/////////////////////////////////////digital output////////////////////////////////////////
G_IO.arDO[5].Ch[0]	:= valve_lift.extend;
G_IO.arDO[5].Ch[1]	:= valve_lift.retract;
G_IO.arDO[5].Ch[2]	:= roller_inbound.roller.forward;
G_IO.arDO[5].Ch[3]	:= roller_inbound.roller.backward;
G_IO.arDO[5].Ch[4]	:= roller_outbound.roller.forward;
G_IO.arDO[5].Ch[5]	:= roller_outbound.roller.backward;
G_IO.arDO[5].Ch[6]	:= roller_outbound_end.roller.forward;
G_IO.arDO[5].Ch[7]	:= roller_outbound_end.roller.backward;
G_IO.arDO[5].Ch[8]	:= lightcurtain_mute_left;
G_IO.arDO[5].Ch[9]	:= lightcurtain_mute_right;

G_IO.arDO[7].Ch[0]	:= valve_vacuun[0].extend;
G_IO.arDO[7].Ch[1]	:= valve_vacuun[1].extend;
G_IO.arDO[7].Ch[2]	:= valve_vacuun[2].extend;
G_IO.arDO[7].Ch[3]	:= valve_vacuun[3].extend;
G_IO.arDO[7].Ch[4]	:= valve_open_side.extend;
G_IO.arDO[7].Ch[8]	:= valve_open_side.retract;
G_IO.arDO[7].Ch[6]	:= valve_open_lift.extend;




/////////////////////////////////////axis config////////////////////////////////////////
mcAxis_lift
(
	ZSN		:=  TRUE OR st_mcAxis_lift.xHoming, //TODO link to digital input
	ZSP		:=  TRUE OR st_mcAxis_lift.xHoming, //TODO link to digital input
	IN_OUT	:= st_mcAxis_lift	, 
	AXIS	:= AxisRef_lift	, 
);
st_mcAxis_lift.bPosSensorShow	:= TRUE;
st_mcAxis_lift.bNegSensorShow	:= TRUE;
st_mcAxis_lift.rMaxAcceleration	:= 50000;
st_mcAxis_lift.rMaxDeceleration	:= 50000;
st_mcAxis_lift.rMaxJerk			:= 500000;
st_mcAxis_lift.rAcceleration	:= 2500;
st_mcAxis_lift.rDeceleration	:= 2500;
st_mcAxis_lift.rJerk			:= 12500;
st_mcAxis_lift.rMaxVelocity		:= 100;
st_mcAxis_lift.rMaxDistance		:= 50;
st_mcAxis_lift.bPosSen	:= TRUE ;//TODO link to digital input
st_mcAxis_lift.bNegSen	:= TRUE ;//TODO link to digital input
st_mcAxis_lift.mcHome.bCalibrationCam	:= TRUE;//TODO link to digital input origin
st_mcAxis_lift.bPositionSensor	:= TRUE;//TODO link to digital input origin
st_mcAxis_lift.bdirFW	:= TRUE;
st_mcAxis_lift.sNetID := '192.168.11.159.5.1';
st_mcAxis_lift.nSlaveAddr	:= 1026;

mcAxis_bag
(
	ZSN		:=  TRUE OR st_mcAxis_bag.xHoming, //TODO link to digital input
	ZSP		:=  TRUE OR st_mcAxis_bag.xHoming, //TODO link to digital input
	IN_OUT	:= st_mcAxis_bag	, 
	AXIS	:= AxisRef_bag	, 
);
st_mcAxis_bag.bPosSensorShow	:= TRUE;
st_mcAxis_bag.bNegSensorShow	:= TRUE;
st_mcAxis_bag.rMaxAcceleration	:= 50000;
st_mcAxis_bag.rMaxDeceleration	:= 50000;
st_mcAxis_bag.rMaxJerk			:= 500000;
st_mcAxis_bag.rAcceleration	:= 2500;
st_mcAxis_bag.rDeceleration	:= 2500;
st_mcAxis_bag.rJerk			:= 12500;
st_mcAxis_bag.rMaxVelocity		:= 100;
st_mcAxis_bag.rMaxDistance		:= 50;
st_mcAxis_bag.bPosSen	:= TRUE ;//TODO link to digital input
st_mcAxis_bag.bNegSen	:= TRUE ;//TODO link to digital input
st_mcAxis_bag.mcHome.bCalibrationCam	:= TRUE;//TODO link to digital input origin
st_mcAxis_bag.bPositionSensor	:= TRUE;//TODO link to digital input origin
st_mcAxis_bag.bdirFW	:= TRUE;
st_mcAxis_bag.sNetID := '192.168.11.159.5.1';
st_mcAxis_bag.nSlaveAddr	:= 1027;

mcAxis_vacuun[0]
(
	ZSN		:=  TRUE OR st_mcAxis_vacuun[0].xHoming, //TODO link to digital input
	ZSP		:=  TRUE OR st_mcAxis_vacuun[0].xHoming, //TODO link to digital input
	IN_OUT	:= st_mcAxis_vacuun[0], 
	AXIS	:= AxisRef_vacuun[0]	, 
);
st_mcAxis_vacuun[0].bPosSensorShow	:= TRUE;
st_mcAxis_vacuun[0].bNegSensorShow	:= TRUE;
st_mcAxis_vacuun[0].rMaxAcceleration	:= 50000;
st_mcAxis_vacuun[0].rMaxDeceleration	:= 50000;
st_mcAxis_vacuun[0].rMaxJerk			:= 500000;
st_mcAxis_vacuun[0].rAcceleration	:= 2500;
st_mcAxis_vacuun[0].rDeceleration	:= 2500;
st_mcAxis_vacuun[0].rJerk			:= 12500;
st_mcAxis_vacuun[0].rMaxVelocity		:= 100;
st_mcAxis_vacuun[0].rMaxDistance		:= 50;
st_mcAxis_vacuun[0].bPosSen	:= TRUE ;//TODO link to digital input
st_mcAxis_vacuun[0].bNegSen	:= TRUE ;//TODO link to digital input
st_mcAxis_vacuun[0].mcHome.bCalibrationCam	:= TRUE;//TODO link to digital input origin
st_mcAxis_vacuun[0].bPositionSensor	:= TRUE;//TODO link to digital input origin
st_mcAxis_vacuun[0].bdirFW	:= TRUE;
st_mcAxis_vacuun[0].sNetID := '192.168.11.159.5.1';
st_mcAxis_vacuun[0].nSlaveAddr	:= 1032;
st_mcAxis_vacuun[0].iAxis	:= 0;

mcAxis_vacuun[1]
(
	ZSN		:=  TRUE OR st_mcAxis_vacuun[1].xHoming, //TODO link to digital input
	ZSP		:=  TRUE OR st_mcAxis_vacuun[1].xHoming, //TODO link to digital input
	IN_OUT	:= st_mcAxis_vacuun[1]	, 
	AXIS	:= AxisRef_vacuun[1]	, 
);
st_mcAxis_vacuun[1].bPosSensorShow	:= TRUE;
st_mcAxis_vacuun[1].bNegSensorShow	:= TRUE;
st_mcAxis_vacuun[1].rMaxAcceleration	:= 50000;
st_mcAxis_vacuun[1].rMaxDeceleration	:= 50000;
st_mcAxis_vacuun[1].rMaxJerk			:= 500000;
st_mcAxis_vacuun[1].rAcceleration	:= 2500;
st_mcAxis_vacuun[1].rDeceleration	:= 2500;
st_mcAxis_vacuun[1].rJerk			:= 12500;
st_mcAxis_vacuun[1].rMaxVelocity		:= 100;
st_mcAxis_vacuun[1].rMaxDistance		:= 50;
st_mcAxis_vacuun[1].bPosSen	:= TRUE ;//TODO link to digital input
st_mcAxis_vacuun[1].bNegSen	:= TRUE ;//TODO link to digital input
st_mcAxis_vacuun[1].mcHome.bCalibrationCam	:= TRUE;//TODO link to digital input origin
st_mcAxis_vacuun[1].bPositionSensor	:= TRUE;//TODO link to digital input origin
st_mcAxis_vacuun[1].bdirFW	:= TRUE;
st_mcAxis_vacuun[1].sNetID := '192.168.11.159.5.1';
st_mcAxis_vacuun[1].nSlaveAddr	:= 1032;
st_mcAxis_vacuun[1].iAxis	:= 1;

mcAxis_bagOpen[0]
(
	ZSN		:=  TRUE OR st_mcAxis_bagOpen[0].xHoming, //TODO link to digital input
	ZSP		:=  TRUE OR st_mcAxis_bagOpen[0].xHoming, //TODO link to digital input
	IN_OUT	:= st_mcAxis_bagOpen[0]	, 
	AXIS	:= AxisRef_bagOpen[0]	, 
);
st_mcAxis_bagOpen[0].bPosSensorShow	:= TRUE;
st_mcAxis_bagOpen[0].bNegSensorShow	:= TRUE;
st_mcAxis_bagOpen[0].rMaxAcceleration	:= 50000;
st_mcAxis_bagOpen[0].rMaxDeceleration	:= 50000;
st_mcAxis_bagOpen[0].rMaxJerk			:= 500000;
st_mcAxis_bagOpen[0].rAcceleration	:= 2500;
st_mcAxis_bagOpen[0].rDeceleration	:= 2500;
st_mcAxis_bagOpen[0].rJerk			:= 12500;
st_mcAxis_bagOpen[0].rMaxVelocity		:= 100;
st_mcAxis_bagOpen[0].rMaxDistance		:= 50;
st_mcAxis_bagOpen[0].bPosSen	:= TRUE ;//TODO link to digital input
st_mcAxis_bagOpen[0].bNegSen	:= TRUE ;//TODO link to digital input
st_mcAxis_bagOpen[0].mcHome.bCalibrationCam	:= TRUE;//TODO link to digital input origin
st_mcAxis_bagOpen[0].bPositionSensor	:= TRUE;//TODO link to digital input origin
st_mcAxis_bagOpen[0].bdirFW	:= TRUE;
st_mcAxis_bagOpen[0].sNetID := '192.168.11.159.5.1';
st_mcAxis_bagOpen[0].nSlaveAddr	:= 1033;
st_mcAxis_bagOpen[0].iAxis	:= 0;

mcAxis_bagOpen[1]
(
	ZSN		:=  TRUE OR st_mcAxis_bagOpen[1].xHoming, //TODO link to digital input
	ZSP		:=  TRUE OR st_mcAxis_bagOpen[1].xHoming, //TODO link to digital input
	IN_OUT	:= st_mcAxis_bagOpen[1]	, 
	AXIS	:= AxisRef_bagOpen[1]	, 
);
st_mcAxis_bagOpen[1].bPosSensorShow	:= TRUE;
st_mcAxis_bagOpen[1].bNegSensorShow	:= TRUE;
st_mcAxis_bagOpen[1].rMaxAcceleration	:= 50000;
st_mcAxis_bagOpen[1].rMaxDeceleration	:= 50000;
st_mcAxis_bagOpen[1].rMaxJerk			:= 500000;
st_mcAxis_bagOpen[1].rAcceleration	:= 2500;
st_mcAxis_bagOpen[1].rDeceleration	:= 2500;
st_mcAxis_bagOpen[1].rJerk			:= 12500;
st_mcAxis_bagOpen[1].rMaxVelocity		:= 100;
st_mcAxis_bagOpen[1].rMaxDistance		:= 50;
st_mcAxis_bagOpen[1].bPosSen	:= TRUE ;//TODO link to digital input
st_mcAxis_bagOpen[1].bNegSen	:= TRUE ;//TODO link to digital input
st_mcAxis_bagOpen[1].mcHome.bCalibrationCam	:= TRUE;//TODO link to digital input origin
st_mcAxis_bagOpen[1].bPositionSensor	:= TRUE;//TODO link to digital input origin
st_mcAxis_bagOpen[1].bdirFW	:= TRUE;
st_mcAxis_bagOpen[1].sNetID := '192.168.11.159.5.1';
st_mcAxis_bagOpen[1].nSlaveAddr	:= 1033;
st_mcAxis_bagOpen[1].iAxis	:= 1;

mcAxis_bagOpen[2]
(
	ZSN		:=  TRUE OR st_mcAxis_bagOpen[2].xHoming, //TODO link to digital input
	ZSP		:=  TRUE OR st_mcAxis_bagOpen[2].xHoming, //TODO link to digital input
	IN_OUT	:= st_mcAxis_bagOpen[2]	, 
	AXIS	:= AxisRef_bagOpen[2]	, 
);
st_mcAxis_bagOpen[2].bPosSensorShow	:= TRUE;
st_mcAxis_bagOpen[2].bNegSensorShow	:= TRUE;
st_mcAxis_bagOpen[2].rMaxAcceleration	:= 50000;
st_mcAxis_bagOpen[2].rMaxDeceleration	:= 50000;
st_mcAxis_bagOpen[2].rMaxJerk			:= 500000;
st_mcAxis_bagOpen[2].rAcceleration	:= 2500;
st_mcAxis_bagOpen[2].rDeceleration	:= 2500;
st_mcAxis_bagOpen[2].rJerk			:= 12500;
st_mcAxis_bagOpen[2].rMaxVelocity		:= 100;
st_mcAxis_bagOpen[2].rMaxDistance		:= 50;
st_mcAxis_bagOpen[2].bPosSen	:= TRUE ;//TODO link to digital input
st_mcAxis_bagOpen[2].bNegSen	:= TRUE ;//TODO link to digital input
st_mcAxis_bagOpen[2].mcHome.bCalibrationCam	:= TRUE;//TODO link to digital input origin
st_mcAxis_bagOpen[2].bPositionSensor	:= TRUE;//TODO link to digital input origin
st_mcAxis_bagOpen[2].bdirFW	:= TRUE;
st_mcAxis_bagOpen[2].sNetID := '192.168.11.159.5.1';
st_mcAxis_bagOpen[2].nSlaveAddr	:= 1034;
st_mcAxis_bagOpen[2].iAxis	:= 0;

mcAxis_bagOpen[3]
(
	ZSN		:=  TRUE OR st_mcAxis_bagOpen[3].xHoming, //TODO link to digital input
	ZSP		:=  TRUE OR st_mcAxis_bagOpen[3].xHoming, //TODO link to digital input
	IN_OUT	:= st_mcAxis_bagOpen[3]	, 
	AXIS	:= AxisRef_bagOpen[3]	, 
);
st_mcAxis_bagOpen[3].bPosSensorShow	:= TRUE;
st_mcAxis_bagOpen[3].bNegSensorShow	:= TRUE;
st_mcAxis_bagOpen[3].rMaxAcceleration	:= 50000;
st_mcAxis_bagOpen[3].rMaxDeceleration	:= 50000;
st_mcAxis_bagOpen[3].rMaxJerk			:= 500000;
st_mcAxis_bagOpen[3].rAcceleration	:= 2500;
st_mcAxis_bagOpen[3].rDeceleration	:= 2500;
st_mcAxis_bagOpen[3].rJerk			:= 12500;
st_mcAxis_bagOpen[3].rMaxVelocity		:= 100;
st_mcAxis_bagOpen[3].rMaxDistance		:= 50;
st_mcAxis_bagOpen[3].bPosSen	:= TRUE ;//TODO link to digital input
st_mcAxis_bagOpen[3].bNegSen	:= TRUE ;//TODO link to digital input
st_mcAxis_bagOpen[3].mcHome.bCalibrationCam	:= TRUE;//TODO link to digital input origin
st_mcAxis_bagOpen[3].bPositionSensor	:= TRUE;//TODO link to digital input origin
st_mcAxis_bagOpen[3].bdirFW	:= TRUE;
st_mcAxis_bagOpen[3].sNetID := '192.168.11.159.5.1';
st_mcAxis_bagOpen[3].nSlaveAddr	:= 1034;
st_mcAxis_bagOpen[3].iAxis	:= 1;



IF MAIN.firstCycle THEN
//	st_mcAxis_bag.mcPower.Enable	:= TRUE;
	st_mcAxis_lift.mcPower.Enable	:= TRUE;	
END_IF
END_METHOD

METHOD M_reset : BOOL
VAR_INPUT
END_VAR
M_reset	:= FALSE;
ton_timeout.IN	:= FALSE;
event.sMethod	:= 'reset';
error_status	:= OrderToteErrorStatus.NO_ERROR;
IF xError THEN
	st_mcAxis_lift.mcStop.Execute	:= FALSE;
	st_mcAxis_vacuun[0].mcStop.Execute	:= FALSE;
	st_mcAxis_vacuun[1].mcStop.Execute	:= FALSE;
	st_mcAxis_bagOpen[0].mcStop.Execute	:= FALSE;
	st_mcAxis_bagOpen[1].mcStop.Execute	:= FALSE;
	st_mcAxis_bagOpen[2].mcStop.Execute	:= FALSE;
	st_mcAxis_bagOpen[3].mcStop.Execute	:= FALSE;	
	st_mcAxis_lift.mcReset.Execute			:= TRUE;
	st_mcAxis_vacuun[0].mcReset.Execute		:= TRUE;
	st_mcAxis_vacuun[1].mcReset.Execute		:= TRUE;
	st_mcAxis_bagOpen[0].mcReset.Execute	:= TRUE;
	st_mcAxis_bagOpen[1].mcReset.Execute	:= TRUE;
	st_mcAxis_bagOpen[2].mcReset.Execute	:= TRUE;
	st_mcAxis_bagOpen[3].mcReset.Execute	:= TRUE;	
	
	IF eStates<>E_WorkingStates.IDLE THEN
		eStates	:= eStateTemp;//continue
	END_IF
		
	xError	:= FALSE;
ELSE
	;
END_IF

//todo:check if reset successful
M_reset	:= TRUE;
END_METHOD

METHOD M_run : BOOL
VAR_INPUT
END_VAR
//
IF M_checkCondition(condition:= E_Condition.NO_TOTE) THEN
	;
END_IF
//check no tote of working
//wait new tote of loading
//tote load
END_METHOD

METHOD M_runStart : BOOL
VAR_INPUT
END_VAR
M_runStart	:= FALSE;

st_mcAxis_vacuun[0].mcPower.Enable	:= TRUE;	
st_mcAxis_vacuun[1].mcPower.Enable	:= TRUE;
st_mcAxis_bagOpen[0].mcPower.Enable	:= TRUE;
st_mcAxis_bagOpen[1].mcPower.Enable	:= TRUE;
st_mcAxis_bagOpen[2].mcPower.Enable	:= TRUE;
st_mcAxis_bagOpen[3].mcPower.Enable	:= TRUE;

st_mcAxis_lift.mcPower.Enable	:= TRUE;

current_tote_status	:= ToteStatus.UNKNOWN;

M_checkCondition(condition:=E_Condition.TOTE_READY);

IF st_mcAxis_vacuun[0].mcReadStatus.StandStill AND st_mcAxis_vacuun[1].mcReadStatus.StandStill AND st_mcAxis_bagOpen[0].mcReadStatus.StandStill
AND st_mcAxis_bagOpen[1].mcReadStatus.StandStill AND st_mcAxis_bagOpen[2].mcReadStatus.StandStill AND st_mcAxis_bagOpen[3].mcReadStatus.StandStill 
AND st_mcAxis_lift.mcReadStatus.StandStill THEN
	M_runStart	:= TRUE;
END_IF	

M_runStart	:= TRUE;
END_METHOD

METHOD M_safetyEvent : BOOL
VAR_INPUT
END_VAR
M_safetyEvent	:= FALSE;

roller_inbound.roller.forward			:= FALSE;
roller_inbound.roller.backward			:= FALSE;
roller_outbound.roller.forward			:= FALSE;
roller_outbound.roller.backward			:= FALSE;
roller_outbound_end.roller.forward		:= FALSE;	
roller_outbound_end.roller.backward		:= FALSE;	

st_mcAxis_vacuun[0].mcMoveAbsolute.Execute	:= FALSE;
st_mcAxis_vacuun[1].mcMoveAbsolute.Execute	:= FALSE;
st_mcAxis_bagOpen[0].mcMoveAbsolute.Execute	:= FALSE;
st_mcAxis_bagOpen[1].mcMoveAbsolute.Execute	:= FALSE;
st_mcAxis_bagOpen[2].mcMoveAbsolute.Execute	:= FALSE;
st_mcAxis_bagOpen[3].mcMoveAbsolute.Execute	:= FALSE;
st_mcAxis_lift.mcMoveAbsolute.Execute	:= FALSE;	

st_mcAxis_vacuun[0].mcStop.Execute	:= TRUE;
st_mcAxis_vacuun[1].mcStop.Execute	:= TRUE;
st_mcAxis_bagOpen[0].mcStop.Execute	:= TRUE;
st_mcAxis_bagOpen[1].mcStop.Execute	:= TRUE;
st_mcAxis_bagOpen[2].mcStop.Execute	:= TRUE;
st_mcAxis_bagOpen[3].mcStop.Execute	:= TRUE;


st_mcAxis_lift.mcStop.Execute	:= TRUE;

M_safetyEvent	:= TRUE;
END_METHOD

METHOD M_toteLoad : BOOL
VAR_INPUT
END_VAR
M_toteLoad	:= FALSE;
IF roller_inbound.photo_sensor.Q THEN
	roller_inbound.roller.forward	:= FALSE;
	ADSLOGSTR(msgCtrlMask:= ADSLOG_MSGTYPE_LOG,msgFmtStr:='tote load finish',strArg:='MSG ARG');
ELSE
	roller_inbound.roller.forward	:= TRUE;
	ADSLOGSTR(msgCtrlMask:= ADSLOG_MSGTYPE_LOG,msgFmtStr:='tote load start',strArg:='MSG ARG');
	M_toteLoad	:= TRUE;
END_IF
END_METHOD

METHOD M_toteUnload : BOOL
VAR_INPUT
END_VAR
M_toteUnload	:= FALSE;

CASE eStates OF 
		E_WorkingStates.TOTE_LIFT_UP:
			valve_lift.extend	:= TRUE;
			valve_lift.retract	:= FALSE;
			IF valve_lift.extended AND NOT valve_lift.retracted THEN
				eStates	:= E_WorkingStates.TOTE_UNLOAD;
			END_IF
		E_WorkingStates.TOTE_OUT:
			IF roller_outbound.photo_sensor.Q THEN
				roller_outbound.roller.forward	:= FALSE;
				M_toteUnload	:= TRUE;
			ELSE
				roller_outbound.roller.forward	:= TRUE;
			END_IF	
		E_WorkingStates.TOTE_LIFT_DOWN:	
			valve_lift.extend	:= FALSE;
			valve_lift.retract	:= TRUE;
			IF NOT valve_lift.extended AND valve_lift.retracted THEN
				M_toteUnload	:= TRUE;
			END_IF	
END_CASE
END_METHOD

METHOD M_unload : BOOL
VAR_INPUT
END_VAR
VAR_OUTPUT 

END_VAR
//initialize
//bag_open lift up & bag_open_home
//tote lift up
//outbound
//tote lift down
//done
M_unload := FALSE;
event.sMethod	:= 'unload';
//////////////////////////////////////////////////////////timeout//////////////////////////////////////////
iStateTemp	:= eStateTemp;
sStateTemp	:= INT_TO_STRING(iStateTemp);
ton_timeout();
IF eStates<>E_WorkingStates.IDLE AND eStates<>E_WorkingStates.ERROR  THEN
	IF eStateTemp=eStates THEN
		ton_timeout.IN	:=TRUE;
	ELSE
		ton_timeout.IN	:=FALSE;
		IF GVL.bAck_stop THEN
			roller_outbound.roller.forward	:= FALSE;
			roller_outbound_end.roller.forward	:= FALSE;
			RETURN;		
		END_IF
		eStateTemp	:= eStates;
	END_IF
ELSE
	ton_timeout.IN	:=FALSE;
END_IF
IF ton_timeout.Q THEN	
	ton_timeout.IN	:=FALSE;
	CASE eStates OF
	
		E_WorkingStates.WAIT_UNLOADING://wait signal from logtech and app to unload the tote
			;
		E_WorkingStates.BAG_OPEN_UP:	
			event.sEventType	:= 'error';
			event.sEvent_MSG	:= CONCAT('BAG_OPEN_UP ','timeout');
			event.sStepID		:= sStateTemp;
		E_WorkingStates.BAG_CLOSE:	
			event.sEventType	:= 'error';
			event.sEvent_MSG	:= CONCAT('BAG_CLOSE or TOTE_LIFT_UP ','timeout');
			event.sStepID		:= sStateTemp;						
		E_WorkingStates.TOTE_LIFT_UP:
			event.sEventType	:= 'error';
			event.sEvent_MSG	:= CONCAT('TOTE_LIFT_UP ','timeout');
			event.sStepID		:= sStateTemp;
		E_WorkingStates.TOTE_UNLOAD:
			event.sEventType	:= 'error';
			event.sEvent_MSG	:= CONCAT('TOTE_UNLOAD ','timeout');
			event.sStepID		:= sStateTemp;

		E_WorkingStates.WAIT_SENSOR_OFF:	
			event.sEventType	:= 'error';
			event.sEvent_MSG	:= CONCAT('WAIT_SENSOR_OFF ','timeout');
			event.sStepID		:= sStateTemp;	
		E_WorkingStates.TOTE_LIFT_DOWN:
			event.sEventType	:= 'error';
			event.sEvent_MSG	:= CONCAT('TOTE_LIFT_DOWN ','timeout');
			event.sStepID		:= sStateTemp;
		ELSE
			event.sEventType	:= 'error';
			event.sEvent_MSG	:= CONCAT('unknow estate ','timeout');
			event.sStepID		:= sStateTemp;			
	END_CASE
	IF eStates<>E_WorkingStates.IDLE AND eStates<>E_WorkingStates.WAIT_UNLOADING AND eStates<>E_WorkingStates.BAG_OPEN_UP THEN
		eStates	:= E_WorkingStates.ERROR;
		error_status	:= OrderToteErrorStatus.MECHANICAL_ERROR;
		Event_add(event);
	END_IF
	
END_IF

CASE eStates OF 
		E_WorkingStates.IDLE:
			
			ton_timeout.PT	:= T#3S;
			xLoading	:= FALSE;
			xUnloading	:= FALSE;
			eStates	:= E_WorkingStates.INIT;
		E_WorkingStates.INIT:	
			ADSLOGSTR(msgCtrlMask:= ADSLOG_MSGTYPE_LOG,msgFmtStr:='unload start',strArg:='');
			xUnloading	:= TRUE;
			st_mcAxis_vacuun[0].mcMoveAbsolute.Execute	:= FALSE;
			st_mcAxis_vacuun[1].mcMoveAbsolute.Execute	:= FALSE;
			st_mcAxis_bagOpen[0].mcMoveAbsolute.Execute	:= FALSE;
			st_mcAxis_bagOpen[1].mcMoveAbsolute.Execute	:= FALSE;
			st_mcAxis_bagOpen[2].mcMoveAbsolute.Execute	:= FALSE;
			st_mcAxis_bagOpen[3].mcMoveAbsolute.Execute	:= FALSE;			
	
			st_mcAxis_lift.mcMoveAbsolute.Execute	:= FALSE;
			eStates	:= E_WorkingStates.WAIT_UNLOADING;
		E_WorkingStates.WAIT_UNLOADING://wait signal from logtech and app to unload the tote
			workflow_status	:= ToteSubsystemWorkflowStatus.WAITING_FOR_UNLOADING;
			tote_status	:= ToteStatus.READY;
			eStates	:= E_WorkingStates.BAG_OPEN_UP;	
			
//		E_WorkingStates.BAG_OPEN_AXIS_CYCLINDER_UP:
//			ton_timeout.PT	:= T#1S;
//			valve_open_lift.extend	:= FALSE;
//			valve_open_lift.retract	:= TRUE;
//			IF NOT valve_open_lift.extended AND valve_open_lift.retracted THEN
//				eStates	:= E_WorkingStates.BAG_OPEN_UP;
//			END_IF
//			IF ton_timeout.Q THEN
//				eStates	:= E_WorkingStates.BAG_OPEN_UP;
//			END_IF
		E_WorkingStates.BAG_OPEN_UP:	
			ton_timeout.PT	:= T#1S;
			valve_open_lift.extend	:= FALSE;
			valve_open_lift.retract	:= TRUE;			
			workflow_status	:= ToteSubsystemWorkflowStatus.OUTBOUNDING;	
			tote_status	:= ToteStatus.LOADED;		
			st_mcAxis_lift.mcMoveAbsolute.Execute	:= TRUE;		
			st_mcAxis_lift.rActualPosSet	:= rPos_lift_up;
			st_mcAxis_lift.rVelocitySet	:= 250;
			IF st_mcAxis_lift.mcMoveAbsolute.Done 
			AND ((NOT valve_open_lift.extended AND valve_open_lift.retracted) OR ton_timeout.Q) THEN
				eStates	:= E_WorkingStates.BAG_OPEN_HOME;
			END_IF	
		E_WorkingStates.BAG_OPEN_HOME:	
			ton_timeout.PT	:= T#5S;
			valve_open_side.extend	:= FALSE;
			valve_open_side.retract	:= TRUE;		
			st_mcAxis_vacuun[0].mcMoveAbsolute.Execute	:= TRUE;		
			st_mcAxis_vacuun[0].rActualPosSet	:= rPos_vacuun_working[0];
			st_mcAxis_vacuun[0].rVelocitySet	:= 450;
			st_mcAxis_vacuun[1].mcMoveAbsolute.Execute	:= TRUE;		
			st_mcAxis_vacuun[1].rActualPosSet	:= rPos_vacuun_working[1];
			st_mcAxis_vacuun[1].rVelocitySet	:= 450;			
			st_mcAxis_bagOpen[0].mcMoveAbsolute.Execute	:= TRUE;		
			st_mcAxis_bagOpen[0].rActualPosSet	:= rPos_bag_begin[0];
			st_mcAxis_bagOpen[0].rVelocitySet	:= 200;			
			st_mcAxis_bagOpen[1].mcMoveAbsolute.Execute	:= TRUE;		
			st_mcAxis_bagOpen[1].rActualPosSet	:= rPos_bag_begin[1];
			st_mcAxis_bagOpen[1].rVelocitySet	:= 200;				
			st_mcAxis_bagOpen[2].mcMoveAbsolute.Execute	:= TRUE;		
			st_mcAxis_bagOpen[2].rActualPosSet	:= rPos_bag_begin[2];
			st_mcAxis_bagOpen[2].rVelocitySet	:= 200;				
			st_mcAxis_bagOpen[3].mcMoveAbsolute.Execute	:= TRUE;		
			st_mcAxis_bagOpen[3].rActualPosSet	:= rPos_bag_begin[3];
			st_mcAxis_bagOpen[3].rVelocitySet	:= 200;		
			valve_lift.extend	:= TRUE;
			valve_lift.retract	:= FALSE;				
			IF st_mcAxis_vacuun[0].mcMoveAbsolute.Done AND st_mcAxis_vacuun[1].mcMoveAbsolute.Done 
			AND st_mcAxis_bagOpen[0].mcMoveAbsolute.Done AND st_mcAxis_bagOpen[1].mcMoveAbsolute.Done 
			AND st_mcAxis_bagOpen[2].mcMoveAbsolute.Done AND st_mcAxis_bagOpen[3].mcMoveAbsolute.Done 
			AND(NOT valve_open_side.extended AND valve_open_side.retracted) 
			AND (valve_lift.extended AND NOT valve_lift.retracted) THEN
				st_mcAxis_vacuun[0].mcMoveAbsolute.Execute	:= FALSE;
				st_mcAxis_vacuun[1].mcMoveAbsolute.Execute	:= FALSE;
				st_mcAxis_bagOpen[0].mcMoveAbsolute.Execute	:= FALSE;
				st_mcAxis_bagOpen[1].mcMoveAbsolute.Execute	:= FALSE;
				st_mcAxis_bagOpen[2].mcMoveAbsolute.Execute	:= FALSE;
				st_mcAxis_bagOpen[3].mcMoveAbsolute.Execute	:= FALSE;
				eStates	:= E_WorkingStates.TOTE_UNLOAD;
			END_IF								
	
//		E_WorkingStates.BAG_CLOSE:	
//			st_mcAxis_bag.mcMoveAbsolute.Execute	:= TRUE;		
//			st_mcAxis_bag.rActualPosSet	:= rPos_bag_closed;
//			st_mcAxis_bag.rVelocitySet	:= 250;
//			valve_lift.extend	:= TRUE;
//			valve_lift.retract	:= FALSE;
//			IF st_mcAxis_bag.mcMoveAbsolute.Done AND valve_lift.extended AND NOT valve_lift.retracted THEN
//				st_mcAxis_bag.mcMoveAbsolute.Execute	:= FALSE;
//				eStates	:= E_WorkingStates.TOTE_UNLOAD;
//			END_IF							
//		E_WorkingStates.TOTE_LIFT_UP:
//			ton_timeout.PT	:= T#3S;
//			valve_lift.extend	:= TRUE;
//			valve_lift.retract	:= FALSE;
//			IF valve_lift.extended AND NOT valve_lift.retracted THEN
//				eStates	:= E_WorkingStates.TOTE_UNLOAD;
//			END_IF
		E_WorkingStates.TOTE_UNLOAD:
			ton_timeout.PT	:= T#5S;
			roller_outbound.roller.forward		:= TRUE;
			roller_outbound_end.roller.forward	:= TRUE;
			IF roller_outbound.photo_sensor.Q THEN
				eStates	:= E_WorkingStates.WAIT_SENSOR_OFF;			
			END_IF	
		E_WorkingStates.WAIT_SENSOR_OFF:
			roller_outbound.roller.forward		:= TRUE;
			roller_outbound_end.roller.forward	:= TRUE;	
			IF NOT roller_outbound.photo_sensor.Q THEN
				roller_outbound.roller.forward		:= FALSE;	
				roller_outbound_end.roller.forward	:= FALSE;
				eStates	:= E_WorkingStates.TOTE_LIFT_DOWN;			
			END_IF			
		E_WorkingStates.TOTE_LIFT_DOWN:
			ton_timeout.PT	:= T#3S;	
			valve_lift.extend	:= FALSE;
			valve_lift.retract	:= TRUE;
			IF NOT valve_lift.extended AND valve_lift.retracted THEN
				eStates	:= E_WorkingStates.DONE;
			END_IF				
		E_WorkingStates.DONE:	
			ADSLOGSTR(msgCtrlMask:= ADSLOG_MSGTYPE_LOG,msgFmtStr:='unload end',strArg:='');
			workflow_status	:= ToteSubsystemWorkflowStatus.IDLE;
			tote_status	:= ToteStatus.EMPTY;			
			M_unload	:= TRUE;
			xUnloading	:= FALSE;
			eStates	:= E_WorkingStates.IDLE;
		E_WorkingStates.ERROR:
			xError	:=	TRUE;
			workflow_status	:= ToteSubsystemWorkflowStatus.IDLE;
			roller_outbound.roller.forward		:= FALSE;	
			roller_outbound_end.roller.forward	:= FALSE;
			st_mcAxis_vacuun[0].mcMoveAbsolute.Execute	:= FALSE;
			st_mcAxis_vacuun[1].mcMoveAbsolute.Execute	:= FALSE;
			st_mcAxis_bagOpen[0].mcMoveAbsolute.Execute	:= FALSE;
			st_mcAxis_bagOpen[1].mcMoveAbsolute.Execute	:= FALSE;
			st_mcAxis_bagOpen[2].mcMoveAbsolute.Execute	:= FALSE;
			st_mcAxis_bagOpen[3].mcMoveAbsolute.Execute	:= FALSE;			
			st_mcAxis_lift.mcMoveAbsolute.Execute	:= FALSE;
			M_unload 		:= TRUE;

		
END_CASE
END_METHOD

METHOD M_waitCondition : BOOL
VAR_INPUT
	condition	: E_Condition;
END_VAR
M_waitCondition	:= FALSE;
CASE condition OF
	E_Condition.NO_TOTE:
	 	IF NOT roller_inbound.photo_sensor.Q THEN
			M_waitCondition	:= TRUE;
		END_IF
	E_Condition.TOTE_IN:
	 	IF roller_inbound.photo_sensor.Q THEN
			M_waitCondition	:= TRUE;
		END_IF	
	E_Condition.READY_LOADING_TOTE:
		IF (pre_tote_status=ToteStatus.READY AND GVL.fb_loading.eTransfer=E_Transfer.UNLOAD) OR tote_status=ToteStatus.LOADED THEN
			M_waitCondition	:= TRUE;
		END_IF	
END_CASE
END_METHOD

END_FUNCTION_BLOCK

// ---- Mian/machine/axis/FB_MotionAxis_MC.TcPOU
FUNCTION_BLOCK FB_MotionAxis_MC

VAR_INPUT
	ZSN	   			: BOOL												;
	ZSP				: BOOL												; 
	Exceeding_us			: INT;
	sNameAxis				: STRING [40];

END_VAR         	
                	
VAR  
	rtFirstCycle	: R_TRIG;						
	mcHomeAxis		: 	MC_HomeAxis						;//ADD BY EVAN 
	sAxisName		: STRING											;//Axis name          	
	xPlus			: BOOL												;	
	xMinus			: BOOL												;
	bDone			: BOOL												;	

// Variables for Hard Stop Homing	                        			
	iStatehsHomig	: E_HomingSteps := E_HomingSteps.IDLE				;
	rtHome			: R_TRIG											;
	rtHomeReset		: R_TRIG											;
	tonTimeOut		: TON												;
	xTimerStart		: BOOL												;
	bLSDefaultVal	: BOOL												; // Save Def value from driver
	xHomeError		: BOOL												;
// Variables for Force Control          					

	rtForceC		: R_TRIG											;
	rtForceCReset	: R_TRIG											;
	DelMaxPos		: LREAL 											;
	rCurrLimit		: LREAL												;
	StartPos		: LREAL												;
	xForceCError	: BOOL												;
//	Variables for Backlash Compensation
	rLastMove		: LREAL := 1										;
	tonBackComp		: TON												;
	rBacklashPer	: LREAL												;	
	
// Variables for errors
	rtError					:	R_TRIG;
	pTextType				:	POINTER TO STRING;
	sAxisErrorID			:	STRING(10);	
	ErrorMSG				:	STRING[255];

//	Exceeding time measuring
	sysTime					:	GETCPUCOUNTER;//GETSYSTEMTIME;					//	Used to measure execution time.
	uStartTime				:	UDINT;
	uFinishTime				:	UDINT;
	ftimeDiff				:	REAL;
	ton_dly	: TON;
	offset	: WORD;
END_VAR         	
                	
VAR_IN_OUT      	
	IN_OUT 			: ST_MotionAxis_MC	;//struct for each axis
	AXIS 			: AXIS_REF			;//Axis obj	
END_VAR

VAR_OUTPUT
	xError			: BOOL				;
	xBusy			: BOOL				;
END_VAR
VAR CONSTANT
	parallelGroupTLName		:	STRING := 'Port_851.TL_Axis_Error';
END_VAR

(* Power options ********************************************************************************************)			
IN_OUT.mcPower(
	Axis				:= AXIS, 
	Enable				:= , 
	Enable_Positive		:= ZSP, 
	Enable_Negative		:= ZSN OR IN_OUT.mcHome.Busy, 
	Override			:= , 
	BufferMode			:= , 
	Options				:= , 
	Status				=> , 
	Busy				=> , 
	Active				=> , 
	Error				=> , 
	ErrorID				=> );
	
(* Halt Mode ********************************************************************************************)	
IN_OUT.mcHalt(
	Axis				:= AXIS, 
	Execute				:= , 
	Deceleration		:= IN_OUT.rDeceleration, 
	Jerk				:= , 
	BufferMode			:= , 
	Options				:= , 
	Done				=> , 
	Busy				=> , 
	Active				=> , 
	CommandAborted		=> , 
	Error				=> , 
	ErrorID				=> );
	
(* Homing ***********************************************************************************************)
IN_OUT.mcHome(
	Axis				:= AXIS, 
	Execute				:= , 
	Position			:= in_out.rFirstpos, 
	HomingMode			:= MC_Direct, 
	BufferMode			:= , 
	Options				:= , 
	bCalibrationCam		:= ,//NOT  ZSN, 
	Done				=> , 
	Busy				=> , 
	Active				=> , 
	CommandAborted		=> , 
	Error				=> , 
	ErrorID				=> );
	
(* JOG **************************************************************************************************)
IN_OUT.mcJog(
	Axis				:= AXIS, 
	JogForward			:= , 
	JogBackwards		:= , 
	Mode				:= E_JogMode.MC_JOGMODE_CONTINOUS, 
	Position			:= , 
	Velocity			:= IN_OUT.rVelocity, 
	Acceleration		:= IN_OUT.rAcceleration, 
	Deceleration		:= IN_OUT.rDeceleration, 
	Jerk				:= IN_OUT.rJerk, 
	Done				=> , 
	Busy				=> , 
	Active				=> , 
	CommandAborted		=> , 
	Error				=> , 
	ErrorID				=> );
	
(* Move Absolute ****************************************************************************************)	
IN_OUT.mcMoveAbsolute(
	Axis				:= AXIS, 
	Execute				:= , 
	Position			:= IN_OUT.rActualPosSet, 
	Velocity			:= IN_OUT.rVelocitySet,     
	Acceleration		:= IN_OUT.rAcceleration, 
	Deceleration		:= IN_OUT.rDeceleration, 
	Jerk				:= IN_OUT.rJerk,         
	BufferMode			:= , 
	Options				:= , 
	Done				=> , 
	Busy				=> , 
	Active				=> , 
	CommandAborted		=> , 
	Error				=> , 
	ErrorID				=> );

	IF IN_OUT.bMoveAbsHMI THEN
		IN_OUT.mcMoveAbsolute.Execute	:= TRUE;
		IN_OUT.rActualPosSet	:= IN_OUT.rActualPosHMI;
		IN_OUT.rVelocitySet		:= IN_OUT.rVeloPers;
	END_IF
(* Move Relative *********************************************************************************************************)
IN_OUT.mcMoveRelative(
	Axis				:= AXIS, 
	Execute				:= , 
	Distance			:= IN_OUT.rPosition + IN_OUT.rBacklashvalue, 
	Velocity			:= IN_OUT.rVelocity,      
	Acceleration		:= IN_OUT.rAcceleration,  
	Deceleration		:= IN_OUT.rDeceleration,  
	Jerk				:= IN_OUT.rJerk,          
	BufferMode			:= ,
	Options				:= , 
	Done				=> bDone, 
	Busy				=> , 
	Active				=> , 
	CommandAborted		=> , 
	Error				=> , 
	ErrorID				=> );
	
(* Move Velocity *********************************************************************************************************)
	
IN_OUT.mcMoveVelocity(
	Axis				:=	AXIS,
	Execute				:=	,
	Velocity			:=	IN_OUT.rVelocity,
	Acceleration		:=	IN_OUT.rAcceleration,
	Deceleration		:=	IN_OUT.rDeceleration,
	Jerk				:=	IN_OUT.rJerk,
	Direction			:=	IN_OUT.axisDirection,
	BufferMode			:=	,
	Options				:=	,
	InVelocity			=>	,
	Busy				=>	,
	Active				=>	,
	CommandAborted		=>	,
	Error				=>	,
	ErrorID				=>	);
	
(**)	
IN_OUT.mcReadStatus(
	Axis				:= AXIS, 
	Enable				:= TRUE, 
	Valid				=> , 
	Busy				=> , 
	Error				=> , 
	ErrorID				=> , 
	ErrorStop			=> , 
	Disabled			=> , 
	Stopping			=> , 
	StandStill			=> , 
	DiscreteMotion		=> , 
	ContinuousMotion	=> , 
	SynchronizedMotion	=> , 
	Homing				=> , 
	ConstantVelocity	=> , 
	Accelerating		=> , 
	Decelerating		=> , 
	Status				=> );
	
(* Reset ************************************************************************************************)
IN_OUT.mcReset(
	Axis				:= AXIS, 
	Execute				:= , 
	Done				=> , 
	Busy				=> , 
	Error				=> , 
	ErrorID				=> );
	
(* Stop *************************************************************************************************)
IN_OUT.mcStop(
	Axis				:= AXIS, 
	Execute				:= , 
	Deceleration		:= , 
	Jerk				:= , 
	Options				:= , 
	Done				=> , 
	Busy				=> , 
	Active				=> , 
	CommandAborted		=> , 
	Error				=> , 
	ErrorID				=> );

(* Set Position *************************************************************************************************)
in_out.mcSetpoint(
	Axis			 := AXIS, 
	Execute			 := , 
	Position		 := IN_OUT.rSetPos, 
	Mode			 := , 
	Options			 := , 
	Done			 => , 
	Busy			 => , 
	Error			 => , 
	ErrorID			 => );


(* write status *************************************************************************************************)
IN_OUT.mcWriteBoolParameter(
	Axis			:= 	AXIS, 
	Execute:= 				, 
	ParameterNumber:= 		, 
	Value:= , 
	Done=> , 
	Busy=> , 
	Error=> , 
	ErrorID=> );

(* Read status *************************************************************************************************)
IN_OUT.mcReadBoolParameter(
	Axis:= AXIS, 
	Enable:= , 
	ParameterNumber:= , 
	ReadMode:= , 
	Valid=> , 
	Busy=> , 
	Error=> , 
	ErrorID=> , 
	Value=> );	

(*Read Actualposition***************************************************************)
IN_OUT.mcReadActualPosition(
	Axis:= AXIS, 
	Enable:= TRUE, 
	Valid=> , 
	Busy=> , 
	Error=> , 
	ErrorID=> , 
	Position=> IN_OUT.rActualPos );   
(*COE write**************************************************************************)	

IN_OUT.CoeWrt(
	sNetId:= IN_OUT.sNetID, 
	nSlaveAddr:= IN_OUT.nSlaveAddr, 
	nSubIndex:= IN_OUT.nSubIndex, 
	nIndex:= IN_OUT.nIndex, 
	pSrcBuf:= ADR(IN_OUT.iSdoWrite), 
	cbBufLen:= SIZEOF(IN_OUT.iSdoWrite), 
	bExecute:= , 
	tTimeout:= , 
	bBusy=> , 
	bError=> , 
	nErrId=> );
	ton_dly(PT:=T#100MS);


offset	:= 16#800*IN_OUT.iAxis;	
CASE IN_OUT.iCoeWrt OF 
	0:
		IN_OUT.CoeWrt.bExecute := FALSE;
	1:
		IN_OUT.CoeWrt.bExecute := TRUE;
		IN_OUT.nIndex	:= 16#2005+offset;
		IN_OUT.nSubIndex	:= 16#1F;
		IN_OUT.iSdoWrite	:= 6;//clear encoder and set current position as origin
		IN_OUT.iCoeWrt	:= 10;
	2:
		IN_OUT.CoeWrt.bExecute := TRUE;
		IN_OUT.nIndex	:= 16#2002+offset;
		IN_OUT.nSubIndex	:= 16#02;
		IN_OUT.iSdoWrite	:= 1;//linear mode
		IN_OUT.iCoeWrt	:= 10;
	3:
		IN_OUT.CoeWrt.bExecute := TRUE;
		IN_OUT.nIndex	:= 16#2002+offset;
		IN_OUT.nSubIndex	:= 16#02;
		IN_OUT.iSdoWrite	:= 2;//rotate mode
		IN_OUT.iCoeWrt	:= 10;
	4:
		IN_OUT.CoeWrt.bExecute := TRUE;
		IN_OUT.nIndex	:= 16#2004+offset;
		IN_OUT.nSubIndex	:= 16#06;
		IN_OUT.iSdoWrite	:= 1;//breaker on
		IN_OUT.iCoeWrt	:= 10;
	5:
		IN_OUT.CoeWrt.bExecute := TRUE;
		IN_OUT.nIndex	:= 16#2004+offset;
		IN_OUT.nSubIndex	:= 16#06;
		IN_OUT.iSdoWrite	:= 0;//breaker off
		IN_OUT.iCoeWrt	:= 10;		
	10:		
		IN_OUT.iCoeWrt	:= 0;
END_CASE







	(*mcHomeAxis***************************************************************)
	mcHomeAxis(
		xExecute:= , 
		xReset:= , 
		InOut:=IN_OUT , 
		xRedy=> , 
		xBusy=> , 
		xDone=> , 
		xError=> ); 
	                                                                                                              	
(******************************************************************************************************************)
	
(**error flag**)

	IN_OUT.xTorqueErr	:=ABS(IN_OUT.rActTorque)>IN_OUT.rToqueLimitSet ;

	
	

	xError := IN_OUT.mcReadStatus.Error OR xHomeError OR IN_OUT.mcMoveAbsolute.Error OR IN_OUT.xTorqueErr ;	
	rtError(CLK:= (IN_OUT.mcReadStatus.ErrorID <> 0 OR xError) AND NOT IN_OUT.xMuteAxisErrorMessages);
	
(*************************** READ ERROR FROM DRIVE *************************)
rtFirstCycle(CLK:= TRUE);
sysTime(cpuCntLoDW => uStartTime);	
sysTime(cpuCntLoDW => uFinishTime);
//M_CheckExceedingTime();

(*************************** GET AXIS ERROR MESSAGE *************************)	
	
	IF rtError.Q THEN
		IF IN_OUT.xTorqueErr THEN
			sAxisErrorID	:= 'TORQUE';
		ELSE
			sAxisErrorID	:=	TO_STRING(IN_OUT.mcReadStatus.ErrorID);
		END_IF
		IN_OUT.mcStop.Execute	:= TRUE;
	
	END_IF
(**remember the Velocity**) 
	IF IN_OUT.rVeloPers <> 0 THEN 
		IN_OUT.rVelocity:= IN_OUT.rVeloPers;
	ELSE 
		IN_OUT.rVeloPers := IN_OUT.rVelocity;	
	END_IF	
(**remember the Acceleration**)
	IF IN_OUT.rAccPers <> 0 THEN 
		IN_OUT.rAcceleration:= IN_OUT.rAccPers;
	ELSE 
		IN_OUT.rAccPers := IN_OUT.rAcceleration;		
	END_IF	
(**remember the Deceleration**)
	IF IN_OUT.rDecPers <> 0 THEN 
		IN_OUT.rDeceleration:= IN_OUT.rDecPers;
	ELSE 
		IN_OUT.rDecPers := IN_OUT.rDeceleration;		
	END_IF
(**False all Executions if function done or error**)
	IF IN_OUT.mcMoveRelative.Done OR IN_OUT.mcMoveRelative.Error OR IN_OUT.mcReset.Busy THEN 
		IN_OUT.mcMoveRelative.Execute := FALSE;
	END_IF

	IF IN_OUT.mcMoveVelocity.Error OR IN_OUT.mcReset.Busy OR IN_OUT.mcMoveVelocity.Busy THEN 
		IN_OUT.mcMoveVelocity.Execute := FALSE;
	END_IF
	
	IF IN_OUT.mcSetpoint.done OR IN_OUT.mcSetpoint.Error THEN
		IN_OUT.mcSetpoint.Execute := FALSE;
	END_IF
	
    IF  IN_OUT.mcMoveAbsolute.Done OR IN_OUT.mcMoveAbsolute.Error OR IN_OUT.mcReset.Busy THEN 
		IN_OUT.mcMoveAbsolute.Execute := FALSE;
	END_IF
 
	 IF IN_OUT.mcHome.Done OR IN_OUT.mcHome.Error THEN 
		IN_OUT.mcHome.Execute := FALSE;
	END_IF
	
	IF IN_OUT.mcStop.Done OR IN_OUT.mcStop.Error THEN 
		IN_OUT.mcStop.Execute := FALSE;
	END_IF
	
	IF IN_OUT.mcReset.Done OR IN_OUT.mcReset.Error THEN 
		IN_OUT.mcReset.Execute := FALSE;
	END_IF
			
	IF IN_OUT.mcReadBoolParameter.Valid OR IN_OUT.mcReadBoolParameter.Error THEN 
		IN_OUT.mcReadBoolParameter.Enable := FALSE;
	END_IF	
	
	IF IN_OUT.mcWriteBoolParameter.Done OR IN_OUT.mcWriteBoolParameter.Error THEN 
		IN_OUT.mcWriteBoolParameter.Execute	:= FALSE;
	END_IF	
		

	
	
	
(**Save done state into temp variable**)	
	
	IF IN_OUT.mcMoveAbsolute.Done THEN
		IN_OUT.xMoveABSDone := TRUE;
	END_IF	
	
	IF IN_OUT.mcMoveRelative.Done THEN
		IN_OUT.xMoveRelDone := TRUE;
	END_IF

PROPERTY P_AxisName : STRING
SET
sAxisName := P_AxisName;
END_SET
END_PROPERTY

PROPERTY P_CurrLimit : LREAL
SET
rCurrLimit := P_CurrLimit;
END_SET
END_PROPERTY

PROPERTY P_DelMaxPos : LREAL
SET
DelMaxPos := P_DelMaxPos;
END_SET
END_PROPERTY

PROPERTY P_ForceCError : BOOL
GET
P_ForceCError := xForceCError;
END_GET
END_PROPERTY

PROPERTY P_hsHomingError : BOOL
GET
P_hsHomingError := xHomeError;
END_GET
END_PROPERTY

PROPERTY P_StartPos : LREAL
SET
StartPos := P_StartPos;
END_SET
END_PROPERTY

END_FUNCTION_BLOCK

// ---- Mian/machine/loading moudle/FB_loading.TcPOU
FUNCTION_BLOCK FB_loading
VAR_INPUT
	pre_tote_status			: ToteStatus;//roller -1 totestatus=ready
	next_tote_status		: ToteStatus;//roller +1 totestatus=empty
	bRun					: BOOL;
	bReset					: BOOL;
	bSafety					: BOOL;
	lightTower				: ST_LightTower;
END_VAR
VAR_OUTPUT
	ready_recive		: BOOL;
	tote_recivied_current		: BOOL;//current roller recived the tote
END_VAR
VAR
	current_tote_status	: ToteStatus;
	ton_timeout			: TON;	
	eStates				: E_LoadingStates := E_LoadingStates.IDLE;
	eStateTemp			: E_LoadingStates := E_LoadingStates.IDLE;
	iStateTemp			: INT;
	sStateTemp			: STRING;
	errorMessage		: STRING;
	xError				: BOOL;
	event				: ST_EVENT;
	rt_error			: R_TRIG;
	eTransfer			: E_Transfer;
///////////////hardware define//////////////////	
	roller_x					: Roller_x;
	roller_y					: Roller_y;
	photo_sensor_tote_detection	: FB_DigitalInput;
	EDM_KA7						: BOOL;
	floodlight					: BOOL;
	mcAxis	 					: FB_MotionAxis_MC;
	st_mcAxis					: ST_MotionAxis_MC;
	AxisRef						: AXIS_REF;	
END_VAR
VAR CONSTANT
	rPos_load	: REAL := 0;
	rPos_unload	: REAL := 1;
	sComponent_name			: STRING := 'fb_loading';
END_VAR

M_mapping();


rt_error(CLK:=(roller_x.roller.err OR roller_y.roller.err OR st_mcAxis.mcReadStatus.Error) 
	AND MAIN.eState<>E_SystemManager.RESET_SAFETY);//roller will trig error while power on
IF rt_error.Q THEN
	xError	:= TRUE;
	eStates	:= E_LoadingStates.ERROR;
END_IF

METHOD M_agingTest : BOOL
VAR_INPUT
	
END_VAR
M_AgingTest	:= FALSE;
//////////////////////////////////////////////////////////timeout//////////////////////////////////////////
iStateTemp	:= eStateTemp;
ton_timeout();
IF eStates<>E_LoadingStates.IDLE AND eStates<>E_LoadingStates.ERROR THEN
	IF eStateTemp=eStates THEN
		ton_timeout.IN	:=TRUE;
	ELSE
		ton_timeout.IN	:=FALSE;
		eStateTemp	:= eStates;
	END_IF
ELSE
	ton_timeout.IN	:=FALSE;
END_IF
IF ton_timeout.Q THEN	
	ton_timeout.IN	:=FALSE;
	CASE eStates OF
		E_LoadingStates.AGING_STATE_0:		
			errorMessage	:= CONCAT('wait loading timeout.->fb_loading ',INT_TO_STRING(iStateTemp));
		E_LoadingStates.AGING_STATE_1:		
			errorMessage	:= CONCAT('wait unloading timeout.->fb_loading ',INT_TO_STRING(iStateTemp));
	END_CASE
	IF eStates<>E_LoadingStates.WAIT AND eStates<>E_LoadingStates.WAIT_1 THEN
		eStates	:= E_LoadingStates.ERROR;
	END_IF
END_IF
CASE eStates OF
	E_LoadingStates.IDLE:
		eStates	:= E_LoadingStates.AGING_STATE_0;
	E_LoadingStates.AGING_STATE_0:
		ton_timeout.PT	:= T#10S;
		roller_x.roller.forward		:= TRUE;
		roller_y.roller.forward		:= TRUE;
		roller_y.roller.backward	:= FALSE;		
		st_mcAxis.mcMoveAbsolute.Execute	:= TRUE;						
		st_mcAxis.rActualPosSet	:= 800;
		st_mcAxis.rVelocitySet	:= 200;
		IF st_mcAxis.mcMoveAbsolute.Done THEN
			eStates	:= E_LoadingStates.WAIT;
		END_IF			
	E_LoadingStates.WAIT:
		roller_x.roller.forward		:= FALSE;
		roller_x.roller.backward	:= FALSE;
		roller_y.roller.forward		:= FALSE;
		roller_y.roller.backward	:= FALSE;	
		st_mcAxis.mcMoveAbsolute.Execute	:= FALSE;
		ton_timeout.PT	:= T#2S;
		IF ton_timeout.Q THEN
			eStates	:= E_LoadingStates.AGING_STATE_1;
		END_IF
	E_LoadingStates.AGING_STATE_1:
		ton_timeout.PT	:= T#10S;
		roller_x.roller.backward	:= TRUE;
		roller_y.roller.forward		:= TRUE;
		roller_y.roller.backward	:= TRUE;			
		st_mcAxis.mcMoveAbsolute.Execute	:= TRUE;						
		st_mcAxis.rActualPosSet	:= 0;
		st_mcAxis.rVelocitySet	:= 200;
		IF st_mcAxis.mcMoveAbsolute.Done THEN
			eStates	:= E_LoadingStates.WAIT_1;
		END_IF	
	E_LoadingStates.WAIT_1:
		roller_x.roller.forward		:= FALSE;
		roller_x.roller.backward	:= FALSE;
		roller_y.roller.forward		:= FALSE;
		roller_y.roller.backward	:= FALSE;	
		st_mcAxis.mcMoveAbsolute.Execute	:= FALSE;	
		ton_timeout.PT	:= T#2S;
		IF ton_timeout.Q THEN
			eStates	:= E_LoadingStates.IDLE;
		END_IF		
	E_LoadingStates.DONE:
		;
	E_LoadingStates.ERROR:
		;
	
END_CASE
END_METHOD

METHOD M_init : BOOL
VAR_INPUT
END_VAR
VAR
END_VAR
M_init	:= FALSE;
xError	:= FALSE;
eStates	:=E_LoadingStates.IDLE;
M_init	:= TRUE;
END_METHOD

METHOD M_load : BOOL
VAR_INPUT
END_VAR
END_METHOD

METHOD M_mapping : BOOL
VAR_INPUT
END_VAR
event.sTime	:= MAIN.Temp_str;
event.sComponent_name	:= sComponent_name;
/////////////////////////////////////digital input////////////////////////////////////////
roller_x.photo_sensor_mute_left(D:= G_IO.arDI[3].Ch[0],on_ms:=10,off_ms:=100);
roller_x.roller.err						:= G_IO.arDI[3].Ch[1];
roller_x.photo_sensor_mute_right(D:= G_IO.arDI[3].Ch[2],on_ms:=10,off_ms:=100);
roller_y.roller.err						:= G_IO.arDI[3].Ch[3];
roller_y.photo_sensor[0](D:= G_IO.arDI[3].Ch[4],on_ms:=100,off_ms:=100);
roller_y.photo_sensor[1](D:= G_IO.arDI[3].Ch[5],on_ms:=100,off_ms:=100);
photo_sensor_tote_detection(D:= G_IO.arDI[3].Ch[6],on_ms:=100,off_ms:=100);
EDM_KA7									:= G_IO.arDI[3].Ch[7];

/////////////////////////////////////digital output////////////////////////////////////////
G_IO.arDO[3].Ch[0]	:= roller_x.roller.forward;
G_IO.arDO[3].Ch[1]	:= roller_x.roller.backward;
G_IO.arDO[3].Ch[2]	:= roller_y.roller.forward;
G_IO.arDO[3].Ch[3]	:= roller_y.roller.backward;
G_IO.arDO[3].Ch[7]	:= lightTower.RED;
G_IO.arDO[3].Ch[8]	:= lightTower.YELLOW;
G_IO.arDO[3].Ch[9]	:= lightTower.GREEN;
G_IO.arDO[3].Ch[10]	:= lightTower.BLUE;
G_IO.arDO[3].Ch[11]	:= lightTower.WHITE;
G_IO.arDO[3].Ch[12]	:= lightTower.BUZZER;
G_IO.arDO[3].Ch[13]	:= floodlight;




/////////////////////////////////////axis config////////////////////////////////////////
mcAxis
(
	ZSN		:=  TRUE OR st_mcAxis.xHoming, //TODO link to digital input
	ZSP		:=  TRUE OR st_mcAxis.xHoming, //TODO link to digital input
	IN_OUT	:= st_mcAxis	, 
	AXIS	:= AxisRef	, 
);
st_mcAxis.bPosSensorShow	:= TRUE;
st_mcAxis.bNegSensorShow	:= TRUE;
st_mcAxis.rMaxAcceleration	:= 50000;
st_mcAxis.rMaxDeceleration	:= 50000;
st_mcAxis.rMaxJerk			:= 500000;
st_mcAxis.rAcceleration	:= 2500;
st_mcAxis.rDeceleration	:= 2500;
st_mcAxis.rJerk			:= 12500;
st_mcAxis.rMaxVelocity		:= 100;
st_mcAxis.rMaxDistance		:= 50;
st_mcAxis.bPosSen	:= TRUE ;//TODO link to digital input
st_mcAxis.bNegSen	:= TRUE ;//TODO link to digital input
st_mcAxis.mcHome.bCalibrationCam	:= TRUE;//TODO link to digital input origin
st_mcAxis.bPositionSensor	:= TRUE;//TODO link to digital input origin
st_mcAxis.bdirFW	:= TRUE;
st_mcAxis.sNetID := '192.168.11.159.5.1';
st_mcAxis.nSlaveAddr	:= 1017;


//
IF MAIN.firstCycle THEN
	st_mcAxis.mcPower.Enable	:= TRUE;
END_IF
END_METHOD

METHOD M_reset : BOOL
VAR_INPUT
END_VAR
M_reset	:= FALSE;
ton_timeout.IN	:= FALSE;
st_mcAxis.mcStop.Execute	:= FALSE;
st_mcAxis.mcReset.Execute	:= TRUE;
IF xError THEN
	IF eStates<>E_LoadingStates.IDLE THEN
		eStates	:= eStateTemp;//continue
	END_IF
	xError	:= FALSE;
ELSE
	M_reset	:= TRUE;
END_IF
END_METHOD

METHOD M_run : BOOL
VAR_INPUT
END_VAR
M_run	:= FALSE;
event.sMethod	:= 'M_run';
//////////////////////////////////////////////////////////current_tote status//////////////////////////////////////////
IF photo_sensor_tote_detection.Q AND NOT(roller_x.photo_sensor_mute_left.Q OR roller_x.photo_sensor_mute_right.Q) THEN
	current_tote_status	:= ToteStatus.READY;
END_IF
IF NOT(roller_x.photo_sensor_mute_left.Q OR roller_x.photo_sensor_mute_right.Q OR photo_sensor_tote_detection.Q
	OR roller_y.photo_sensor[0].Q OR roller_y.photo_sensor[1].Q OR roller_y.roller.sensor.Q) THEN
	current_tote_status	:= ToteStatus.EMPTY;
END_IF
//////////////////////////////////////////////////////////timeout//////////////////////////////////////////
IF 	eStates=E_LoadingStates.LIFT_POSITION_UNLOAD
	OR eStates=	E_LoadingStates.ROLLER_UNLOAD		
	OR eStates=	E_LoadingStates.WAIT_RIGHT_MUTE_OFF THEN
	IF MAIN.application.tote_subsystem.cmd<>OrderToteCommand.LOAD THEN//not count timer and run until cmd=load
		RETURN;
	END_IF
END_IF
		
		
iStateTemp	:= eStateTemp;
sStateTemp	:= INT_TO_STRING(iStateTemp);
ton_timeout();
IF eStates<>E_LoadingStates.IDLE AND eStates<>E_LoadingStates.ERROR THEN
	IF eStateTemp=eStates THEN
		ton_timeout.IN	:=TRUE;
	ELSE
		ton_timeout.IN	:=FALSE;
		IF GVL.bAck_stop THEN
			roller_x.roller.forward	:= FALSE;
			RETURN;		
		END_IF
		eStateTemp	:= eStates;
	END_IF
ELSE
	ton_timeout.IN	:=FALSE;
END_IF
IF ton_timeout.Q THEN	
	ton_timeout.IN	:=FALSE;
	CASE eStates OF		
		E_LoadingStates.LOADING:	
			event.sEventType	:= 'error';
			event.sEvent_MSG	:=  CONCAT('LOADING ','timeout');
			event.sStepID		:= sStateTemp;
		E_LoadingStates.LIFT_POSITION_LOAD:		
			event.sEventType	:= 'error';
			event.sEvent_MSG	:=  CONCAT('LIFT_POSITION_LOAD ','timeout');
			event.sStepID		:= sStateTemp;
		E_LoadingStates.ROLLER_LOAD:
			event.sEventType	:= 'error';
			event.sEvent_MSG	:=  CONCAT('ROLLER_LOAD ','timeout');
			event.sStepID		:= sStateTemp;
		E_LoadingStates.WAIT_LEFT_MUTE_OFF:
			event.sEventType	:= 'error';
			event.sEvent_MSG	:=  CONCAT('WAIT_LEFT_MUTE_OFF ','timeout');
			event.sStepID		:= sStateTemp;
		E_LoadingStates.UNLOADING:	
			event.sEventType	:= 'error';
			event.sEvent_MSG	:=  CONCAT('UNLOADING ','timeout');
			event.sStepID		:= sStateTemp;
		E_LoadingStates.LIFT_POSITION_UNLOAD:	
			event.sEventType	:= 'error';
			event.sEvent_MSG	:=  CONCAT('LIFT_POSITION_UNLOAD ','timeout');
			event.sStepID		:= sStateTemp;
		E_LoadingStates.ROLLER_UNLOAD:
			event.sEventType	:= 'error';
			event.sEvent_MSG	:=  CONCAT('ROLLER_UNLOAD ','timeout');
			event.sStepID		:= sStateTemp;	
		E_LoadingStates.WAIT_RIGHT_MUTE_OFF:
			event.sEventType	:= 'error';
			event.sEvent_MSG	:=  CONCAT('WAIT_RIGHT_MUTE_OFF ','timeout');
			event.sStepID		:= sStateTemp;	
	END_CASE
	IF eStates<>E_LoadingStates.WAIT AND eStates<>E_LoadingStates.DETECTION AND eStates<>E_LoadingStates.WAIT_NEXT_READY THEN
		eStates	:= E_LoadingStates.ERROR;
		Event_add(event);
	END_IF
END_IF

CASE eStates OF 
		E_LoadingStates.IDLE:	
			eStates	:= E_LoadingStates.INIT;
		E_LoadingStates.INIT:
			eStates	:= E_LoadingStates.WAIT;
		E_LoadingStates.WAIT:
			eStates	:= E_LoadingStates.DETECTION;
		E_LoadingStates.DETECTION:
			st_mcAxis.mcMoveAbsolute.Execute	:= FALSE;
			roller_x.roller.forward	:= FALSE;
			ton_timeout.PT	:= T#10S;
			eTransfer	:= E_Transfer.IDLE;
			IF current_tote_status=ToteStatus.EMPTY AND pre_tote_status=ToteStatus.READY THEN
				eStates	:= E_LoadingStates.LOADING;
			END_IF
			IF next_tote_status=ToteStatus.EMPTY AND current_tote_status=ToteStatus.READY AND MAIN.application.tote_subsystem.cmd=OrderToteCommand.LOAD THEN
				eStates	:= E_LoadingStates.UNLOADING;
			END_IF				
		E_LoadingStates.LOADING:	
			eStates	:= E_LoadingStates.LIFT_POSITION_LOAD;
		E_LoadingStates.LIFT_POSITION_LOAD:				
			st_mcAxis.mcMoveAbsolute.Execute	:= TRUE;						
			st_mcAxis.rActualPosSet	:= rPos_load;
			st_mcAxis.rVelocitySet	:= 100;
			IF st_mcAxis.mcMoveAbsolute.Done THEN
				st_mcAxis.mcMoveAbsolute.Execute	:= FALSE;
				eTransfer	:= E_Transfer.LOAD;
				eStates	:= E_LoadingStates.ROLLER_LOAD;
			END_IF	
		E_LoadingStates.ROLLER_LOAD:
			roller_x.roller.forward	:= TRUE;
			IF photo_sensor_tote_detection.Q THEN
				eStates	:= E_LoadingStates.WAIT_LEFT_MUTE_OFF;
			END_IF
		E_LoadingStates.WAIT_LEFT_MUTE_OFF:
			roller_x.roller.forward	:= TRUE;
			IF NOT roller_x.photo_sensor_mute_left.Q THEN
				roller_x.roller.forward	:= FALSE;
				eStates	:= E_LoadingStates.DETECTION;
			END_IF	
		E_LoadingStates.UNLOADING:	
			eStates	:= E_LoadingStates.LIFT_POSITION_UNLOAD;
		E_LoadingStates.LIFT_POSITION_UNLOAD:
			st_mcAxis.mcMoveAbsolute.Execute	:= TRUE;						
			st_mcAxis.rActualPosSet	:= rPos_unload;
			st_mcAxis.rVelocitySet	:= 100;
			IF st_mcAxis.mcMoveAbsolute.Done THEN
				st_mcAxis.mcMoveAbsolute.Execute	:= FALSE;
				eStates	:= E_LoadingStates.WAIT_NEXT_READY;
			END_IF	
		E_LoadingStates.WAIT_NEXT_READY:
			eTransfer	:= E_Transfer.UNLOAD;
			IF GVL.fb_working.eStates=E_WorkingStates.TOTE_LOAD THEN
				eStates	:= E_LoadingStates.ROLLER_UNLOAD;
			END_IF			
		E_LoadingStates.ROLLER_UNLOAD:
			roller_x.roller.forward	:= TRUE;
			IF NOT photo_sensor_tote_detection.Q THEN
				eStates	:= E_LoadingStates.WAIT_RIGHT_MUTE_OFF;
			END_IF			
		E_LoadingStates.WAIT_RIGHT_MUTE_OFF:
			roller_x.roller.forward	:= TRUE;
			IF NOT roller_x.photo_sensor_mute_right.Q THEN
				roller_x.roller.forward	:= FALSE;
				eStates	:= E_LoadingStates.DETECTION;
			END_IF				
		E_LoadingStates.DONE:			
			eStates	:= E_LoadingStates.IDLE;
		E_LoadingStates.ERROR:
			st_mcAxis.mcMoveAbsolute.Execute	:= FALSE;
			roller_x.roller.forward	:= FALSE;			
			xError	:=	TRUE;	
END_CASE
END_METHOD

METHOD M_runStart : BOOL
VAR_INPUT
END_VAR
M_runStart	:= FALSE;
st_mcAxis.mcPower.Enable	:= TRUE;
IF st_mcAxis.mcReadStatus.StandStill THEN
	M_runStart	:= TRUE;
END_IF
M_runStart	:= TRUE;
END_METHOD

METHOD M_safetyEvent : BOOL
VAR_INPUT
END_VAR
M_safetyEvent	:= FALSE;

roller_x.roller.forward		:= FALSE;
roller_x.roller.backward	:= FALSE;
roller_y.roller.forward		:= FALSE;
roller_y.roller.backward	:= FALSE;
st_mcAxis.mcMoveAbsolute.Execute	:= FALSE;
st_mcAxis.mcStop.Execute	:= TRUE;

M_safetyEvent	:= TRUE;
END_METHOD

METHOD M_unload : BOOL
VAR_INPUT
END_VAR
END_METHOD

END_FUNCTION_BLOCK

// ---- Mian/Event_add.TcPOU
FUNCTION Event_add : BOOL
VAR_INPUT
	event	: ST_EVENT;
END_VAR
VAR
	i :INT;
END_VAR

//write event
FOR i:=0 TO GVL.iAlarm_max DO
	IF GVL.events_alarm[i].sEvent_MSG='' THEN
		GVL.events_alarm[i]	:= event;
		EXIT;
	END_IF
END_FOR
//check full
IF GVL.events_alarm[GVL.iAlarm_max].sEvent_MSG<>'' THEN
	FOR i:=0 TO GVL.iAlarm_max-1 DO
		GVL.events_alarm[i]	:= GVL.events_alarm[i+1];
	END_FOR
	GVL.events_alarm[GVL.iAlarm_max]	:= GVL.event_for_clear;
END_IF

END_FUNCTION

// ---- Mian/machine/bufferr module/FB_buffer.TcPOU
FUNCTION_BLOCK FB_buffer
VAR_INPUT
END_VAR
VAR_OUTPUT
END_VAR
VAR

	fb_rollers		: ARRAY[0..iHas_rollers] OF FB_roller;
	sensor_start	: ARRAY[0..1] OF FB_DigitalInput;//sensor at the beginning of roller[0]
	EDM_24v	: BOOL;//edm_24v
	EDM_sto	: BOOL;//edm_sto
	xError	: BOOL;
	
	i	: INT;
	event				: ST_EVENT;
	rt_error			: R_TRIG;
	bStopped			: BOOL;
END_VAR
VAR CONSTANT
	iHas_rollers	: INT:=3;
	sComponent_name			: STRING := 'fb_buffer';
END_VAR

M_mapping();
event.sTime	:= MAIN.Temp_str;
event.sComponent_name	:= sComponent_name;
xError	:= fb_rollers[0].xError OR fb_rollers[1].xError OR fb_rollers[2].xError  OR fb_rollers[3].xError;
		
bstopped	:= fb_rollers[0].bStopped AND fb_rollers[1].bStopped AND fb_rollers[2].bStopped AND fb_rollers[3].bStopped;

METHOD M_agingTest : BOOL
VAR_INPUT
END_VAR
FOR i:=0 TO iHas_rollers DO
	fb_rollers[i].M_agingTest();
END_FOR
END_METHOD

METHOD M_init : BOOL
VAR_INPUT
END_VAR
VAR
	i: INT;
END_VAR
M_init	:= FALSE;

FOR i:=0 TO iHas_rollers DO
	fb_rollers[i].M_init();
END_FOR
xError	:= FALSE;
M_init	:= TRUE;
END_METHOD

METHOD M_mapping : BOOL
VAR_INPUT
END_VAR

//todo:reconfig dios
/////////////////////////////////////digital input////////////////////////////////////////

fb_rollers[0].roller.err			:= G_IO.arDI[1].Ch[0];
fb_rollers[1].roller.err			:= G_IO.arDI[1].Ch[1];
fb_rollers[1].roller.sensor(D:= G_IO.arDI[1].Ch[2],on_ms:=100,off_ms:=100);
fb_rollers[2].roller.sensor(D:= G_IO.arDI[1].Ch[3],on_ms:=100,off_ms:=100);
fb_rollers[2].roller.err			:= G_IO.arDI[1].Ch[4];
fb_rollers[3].roller.err			:= G_IO.arDI[1].Ch[5];
fb_rollers[3].roller.sensor(D:= G_IO.arDI[1].Ch[6],on_ms:=100,off_ms:=100);
fb_rollers[3].sensor_mute(D:= G_IO.arDI[1].Ch[7],on_ms:=10,off_ms:=100);
EDM_24v								:= G_IO.arDI[1].Ch[11];
EDM_sto								:= G_IO.arDI[1].Ch[12];
sensor_start[0](D:= G_IO.arDI[1].Ch[13],on_ms:=100,off_ms:=100);
sensor_start[1](D:= G_IO.arDI[1].Ch[15],on_ms:=100,off_ms:=100);
fb_rollers[0].roller.sensor(D:= G_IO.arDI[1].Ch[14],on_ms:=100,off_ms:=100);

/////////////////////////////////////digital output////////////////////////////////////////
G_IO.arDO[1].Ch[0]	:= fb_rollers[2].roller.forward;
G_IO.arDO[1].Ch[1]	:= fb_rollers[2].roller.backward;
G_IO.arDO[1].Ch[2]	:= fb_rollers[0].roller.forward;
G_IO.arDO[1].Ch[3]	:= fb_rollers[0].roller.backward;
G_IO.arDO[1].Ch[4]	:= fb_rollers[1].roller.forward;
G_IO.arDO[1].Ch[5]	:= fb_rollers[1].roller.backward;
G_IO.arDO[1].Ch[6]	:= fb_rollers[3].roller.forward;
G_IO.arDO[1].Ch[7]	:= fb_rollers[3].roller.backward;



/////////////////////////////////////fb rollers////////////////////////////////////////

FOR i:=0 TO iHas_rollers DO
	fb_rollers[i].M_mapping(i);
END_FOR
END_METHOD

METHOD M_reset : BOOL
VAR_INPUT
END_VAR

VAR
	i: INT;
END_VAR
M_reset	:= FALSE;

FOR i:=0 TO iHas_rollers DO
	IF fb_rollers[i].M_reset() THEN
		CONTINUE;
	END_IF
END_FOR

M_reset	:= TRUE;
END_METHOD

METHOD M_run : BOOL
VAR_INPUT
END_VAR
M_run	:= FALSE;
IF sensor_start[0].Q OR sensor_start[1].Q THEN
	fb_rollers[0].pre_tote_status := ToteStatus.READY;
ELSE
	fb_rollers[0].pre_tote_status := ToteStatus.EMPTY;
END_IF
fb_rollers[0](	id_roller := 0,
				next_tote_status := fb_rollers[1].current_tote_status);
fb_rollers[1](	id_roller := 1,
				pre_tote_status := fb_rollers[0].current_tote_status,
				next_tote_status := fb_rollers[2].current_tote_status);
fb_rollers[2](	id_roller := 2,
				pre_tote_status := fb_rollers[1].current_tote_status,
				next_tote_status := fb_rollers[3].current_tote_status);
fb_rollers[3](	id_roller := 3,
				pre_tote_status := fb_rollers[2].current_tote_status,
				next_tote_status := GVL.fb_loading.current_tote_status);
END_METHOD

METHOD M_runStart : BOOL
VAR_INPUT
END_VAR
VAR
	pSt_mcAxis	:POINTER TO ST_MotionAxis_MC;
END_VAR
M_runStart	:= FALSE;
pSt_mcAxis	:= ADR(fb_rollers[3].st_mcAxis);
pSt_mcAxis^.mcPower.Enable	:= TRUE;
IF pSt_mcAxis^.mcReadStatus.StandStill THEN
	M_runStart	:= TRUE;
END_IF
END_METHOD

METHOD M_safetyEvent : BOOL
VAR_INPUT
END_VAR
FOR i:=0 TO iHas_rollers DO
	fb_rollers[i].M_safetyEvent();
END_FOR
END_METHOD

END_FUNCTION_BLOCK

// ---- Mian/machine/bufferr module/FB_roller.TcPOU
FUNCTION_BLOCK FB_roller
VAR_INPUT
	pre_tote_status			: ToteStatus;//roller -1 totestatus=ready
	next_tote_status		: ToteStatus;//roller +1 totestatus=empty
	roller					: Roller;	
	id_roller				: INT;
	sensor_mute				: FB_DigitalInput;
END_VAR
VAR_OUTPUT
	
END_VAR
VAR_IN_OUT
	
END_VAR
	
VAR
	mcAxis			: FB_MotionAxis_MC;
	st_mcAxis 		: ST_MotionAxis_MC;
	AxisRef			: AXIS_REF;
	current_tote_status		: ToteStatus;//state of current roller tote
	ton_timeout	: TON;	
	eStates					: E_RollerStates :=	E_RollerStates.IDLE;
	eStateTemp				: E_RollerStates :=	E_RollerStates.IDLE;
	iStateTemp				: INT;
	sStateTemp				: STRING;
	errorMessage			: STRING;
	xError	: BOOL;
	event				: ST_EVENT;
	rt_error			: R_TRIG;
	bStopped				: BOOL;
	rTrig_addEvent	:ARRAY[0..10] OF R_TRIG;
END_VAR
VAR CONSTANT
	rPos_up			: REAL	:=90;
	rPos_down			: REAL	:=0;
	sComponent_name			: STRING := 'fb_roller';
END_VAR


//////////////////////////////////////////////////////////timeout//////////////////////////////////////////
iStateTemp	:= eStateTemp;
sStateTemp	:= INT_TO_STRING(iStateTemp);
ton_timeout();
IF eStates<>E_RollerStates.IDLE AND eStates<>E_RollerStates.ERROR THEN
	IF eStateTemp=eStates THEN
		ton_timeout.IN	:=TRUE;
	ELSE
		ton_timeout.IN	:=FALSE;
		IF GVL.bAck_pause THEN
			RETURN;		
		END_IF		
		eStateTemp	:= eStates;
	END_IF
ELSE
	ton_timeout.IN	:=FALSE;
END_IF
IF ton_timeout.Q THEN	
	ton_timeout.IN	:=FALSE;
	CASE eStates OF
		E_RollerStates.STOPPER_DOWN:		
			event.sEventType	:= 'error';
			event.sEvent_MSG	:=  CONCAT('STOPPER_DOWN ','timeout');
			event.sStepID		:=	sStateTemp;
		E_RollerStates.ROLLER_UNLOAD:		
			event.sEventType	:= 'error';
			event.sEvent_MSG	:=  CONCAT('ROLLER_UNLOAD ','timeout');
			event.sStepID		:=  sStateTemp;
		E_RollerStates.WAIT_MUTE_OFF:
			event.sEventType	:= 'error';
			event.sEvent_MSG	:=  CONCAT('WAIT_MUTE_OFF ','timeout');
			event.sStepID		:=  sStateTemp;
		E_RollerStates.STOPPER_UP:			
			event.sEventType	:= 'error';
			event.sEvent_MSG	:=  CONCAT('STOPPER_UP ','timeout');
			event.sStepID		:=  sStateTemp;						
	END_CASE
	IF eStates<>E_RollerStates.DETECTION AND eStates<>E_RollerStates.LOADING AND eStates<>E_RollerStates.UNLOADING THEN
		eStates	:= E_RollerStates.ERROR;
		Event_add(event);
	END_IF
END_IF

CASE eStates OF 
		E_RollerStates.IDLE:
			roller.forward	:= FALSE;
			IF NOT GVL.bAck_stop THEN
				eStates	:= E_RollerStates.INIT;
			END_IF
		E_RollerStates.INIT:	
			ton_timeout.PT	:= T#10S;
			eStates	:= E_RollerStates.DETECTION;
		E_RollerStates.DETECTION:
			roller.forward	:= FALSE;
			st_mcAxis.mcMoveAbsolute.Execute	:= FALSE;		
			IF roller.sensor.Q THEN
				current_tote_status	:= ToteStatus.READY;
			ELSE
				current_tote_status	:= ToteStatus.EMPTY;
			END_IF		
			IF pre_tote_status=ToteStatus.READY AND current_tote_status=ToteStatus.EMPTY THEN
				eStates	:= E_RollerStates.LOADING;
			END_IF
			IF next_tote_status=ToteStatus.EMPTY AND current_tote_status=ToteStatus.READY THEN
				IF id_roller=3 THEN
					IF GVL.fb_loading.eTransfer=E_Transfer.LOAD THEN
						eStates	:= E_RollerStates.UNLOADING;
					END_IF
				ELSE
					eStates	:= E_RollerStates.UNLOADING;
				END_IF					
			END_IF
			IF GVL.bAck_stop THEN
				eStates	:= E_RollerStates.IDLE;
			END_IF
///////////////////////////////load/////////////////////////////////			
		E_RollerStates.LOADING:	
			current_tote_status	:= ToteStatus.UNKNOWN;	
			IF roller.sensor.Q THEN
				eStates	:= E_RollerStates.DONE;
				roller.forward	:= FALSE;
			ELSE
				roller.forward	:= TRUE;
			END_IF
			IF ton_timeout.Q THEN
				eStates	:= E_RollerStates.DONE;
			END_IF
///////////////////////////////unload/////////////////////////////////
		E_RollerStates.UNLOADING:
			current_tote_status	:= ToteStatus.UNKNOWN;	
			IF id_roller=3 THEN
				eStates	:= E_RollerStates.STOPPER_DOWN;
			ELSE	
				IF roller.sensor.Q THEN			
					roller.forward	:= TRUE;
				ELSE
					eStates	:= E_RollerStates.DONE;
					roller.forward	:= FALSE;
				END_IF	
				IF ton_timeout.Q THEN
					eStates	:= E_RollerStates.DONE;
				END_IF
			END_IF	
		E_RollerStates.STOPPER_DOWN:
			st_mcAxis.mcMoveAbsolute.Execute	:= TRUE;						
			st_mcAxis.rActualPosSet	:= rPos_down;
			st_mcAxis.rVelocitySet	:= 100;
			IF st_mcAxis.mcMoveAbsolute.Done THEN
				st_mcAxis.mcMoveAbsolute.Execute	:= FALSE;
				eStates	:= E_RollerStates.ROLLER_UNLOAD;
			END_IF					
		E_RollerStates.ROLLER_UNLOAD:
			roller.forward	:= TRUE;
			IF sensor_mute.Q THEN
				eStates	:= E_RollerStates.WAIT_MUTE_OFF;
			END_IF
		E_RollerStates.WAIT_MUTE_OFF:
			IF NOT sensor_mute.Q THEN
				roller.forward	:= FALSE;
				eStates	:= E_RollerStates.STOPPER_UP;
			END_IF
		E_RollerStates.STOPPER_UP:
			st_mcAxis.mcMoveAbsolute.Execute	:= TRUE;						
			st_mcAxis.rActualPosSet	:= rPos_up;
			st_mcAxis.rVelocitySet	:= 100;
			IF st_mcAxis.mcMoveAbsolute.Done THEN
				st_mcAxis.mcMoveAbsolute.Execute	:= FALSE;
				eStates	:= E_RollerStates.DONE;
			END_IF			
		E_RollerStates.DONE:			
			eStates	:= E_RollerStates.IDLE;
		E_RollerStates.ERROR:
			st_mcAxis.mcMoveAbsolute.Execute	:= FALSE;
			roller.forward	:= FALSE;
			xError	:=	TRUE;	
END_CASE

////////////////////////////////////////////////////////////////////////////////////////////////////
M_mapping(id_roller);

IF eStates=E_RollerStates.IDLE OR MAIN.eState<>E_SystemManager.IN_PROGRESS THEN
	bStopped	:= TRUE;
ELSE
	bStopped	:= FALSE;
END_IF 
//////////////////////////////////////////electrical error///////////////////////////////////////////////
rt_error(CLK:=(roller.err OR st_mcAxis.mcReadStatus.Error)AND MAIN.eState<>E_SystemManager.RESET_SAFETY);//roller will trig error while power on

IF rt_error.Q THEN
	xError	:= TRUE;
	eStates	:= E_RollerStates.ERROR;
END_IF
//////////////////////////////////////////write electrical error///////////////////////////////////////////////
rTrig_addEvent[0](CLK:=roller.err);
rTrig_addEvent[1](CLK:=id_roller=3 AND st_mcAxis.mcReadStatus.Error);
IF MAIN.eState<>E_SystemManager.RESET_SAFETY AND MAIN.eState<>E_SystemManager.RESET_FB_LOADING THEN
	IF rTrig_addEvent[0].Q THEN
		event.sEventType	:= 'ELECTRICAL ERROR';
		event.sEvent_MSG	:= 'roller is in error state';
		Event_add(event);		
	END_IF
	IF rTrig_addEvent[1].Q THEN
		event.sEventType	:= 'ELECTRICAL ERROR';
		event.sEvent_MSG	:= 'axis of stopper is in error state';
		Event_add(event);		
	END_IF		
END_IF

METHOD M_agingTest : BOOL
VAR_INPUT
END_VAR
M_AgingTest	:= FALSE;
//////////////////////////////////////////////////////////timeout//////////////////////////////////////////
iStateTemp	:= eStateTemp;
ton_timeout();
IF eStates<>E_RollerStates.IDLE AND eStates<>E_RollerStates.ERROR THEN
	IF eStateTemp=eStates THEN
		ton_timeout.IN	:=TRUE;
	ELSE
		ton_timeout.IN	:=FALSE;
		eStateTemp	:= eStates;
	END_IF
ELSE
	ton_timeout.IN	:=FALSE;
END_IF
IF ton_timeout.Q THEN	
	ton_timeout.IN	:=FALSE;
	CASE eStates OF
		E_RollerStates.AGING_STATE_0:		
			errorMessage	:= CONCAT('wait loading timeout.->fb_loading ',INT_TO_STRING(iStateTemp));
		E_RollerStates.AGING_STATE_1:		
			errorMessage	:= CONCAT('wait unloading timeout.->fb_loading ',INT_TO_STRING(iStateTemp));
	END_CASE
	IF eStates<>E_RollerStates.WAIT AND eStates<>E_RollerStates.WAIT_1 THEN
		//eStates	:= E_RollerStates.ERROR;
		;
	END_IF
END_IF
CASE eStates OF
	E_RollerStates.IDLE:
		eStates	:= E_RollerStates.AGING_STATE_0;
	E_RollerStates.AGING_STATE_0:
		ton_timeout.PT	:= T#5S;
		roller.forward	:= TRUE;
		roller.backward	:= FALSE;
		st_mcAxis.mcMoveAbsolute.Execute	:= TRUE;						
		st_mcAxis.rActualPosSet	:= rPos_up;
		st_mcAxis.rVelocitySet	:= 100;
		//IF st_mcAxis.mcMoveAbsolute.Done AND ton_timeout.Q THEN
		IF ton_timeout.Q THEN	
			eStates	:= E_RollerStates.WAIT;
		END_IF			
	E_RollerStates.WAIT:
		roller.forward			:= FALSE;
		roller.backward			:= FALSE;	
		st_mcAxis.mcMoveAbsolute.Execute	:= FALSE;	
		ton_timeout.PT	:= T#2S;
		IF ton_timeout.Q THEN
			eStates	:= E_RollerStates.AGING_STATE_1;
		END_IF
	E_RollerStates.AGING_STATE_1:
		ton_timeout.PT	:= T#5S;
		roller.forward	:= TRUE;
		roller.backward	:= TRUE;
		st_mcAxis.mcMoveAbsolute.Execute	:= TRUE;						
		st_mcAxis.rActualPosSet	:= rPos_down;
		st_mcAxis.rVelocitySet	:= 100;
		//IF st_mcAxis.mcMoveAbsolute.Done AND ton_timeout.Q THEN
		IF ton_timeout.Q THEN	
			eStates	:= E_RollerStates.WAIT_1;
		END_IF	
	E_RollerStates.WAIT_1:
		roller.forward			:= FALSE;
		roller.backward			:= FALSE;	
		st_mcAxis.mcMoveAbsolute.Execute	:= FALSE;	
		ton_timeout.PT	:= T#2S;
		IF ton_timeout.Q THEN
			eStates	:= E_RollerStates.IDLE;
		END_IF	
	E_RollerStates.DONE:
		;
	E_RollerStates.ERROR:
		;
	
END_CASE
END_METHOD

METHOD M_init : BOOL
VAR_INPUT
END_VAR
VAR
END_VAR
M_init	:= FALSE;
eStates	:=E_RollerStates.IDLE;
xError	:= FALSE;
st_mcAxis.mcStop.Execute	:= FALSE;
st_mcAxis.mcReset.Execute	:= TRUE;


M_init	:= TRUE;
END_METHOD

METHOD M_mapping : BOOL
VAR_INPUT
	i	: INT;
END_VAR
event.sTime	:= MAIN.Temp_str;
event.sComponent_name	:= sComponent_name;
event.sComponentID	:= INT_TO_STRING(id_roller);
/////////////////////
mcAxis
(
	ZSN		:=  TRUE OR st_mcAxis.xHoming, //TODO link to digital input
	ZSP		:=  TRUE OR st_mcAxis.xHoming, //TODO link to digital input
	IN_OUT	:= 	st_mcAxis, 
	AXIS	:= 	AxisRef	, 
);
st_mcAxis.bPosSensorShow	:= TRUE;
st_mcAxis.bNegSensorShow	:= TRUE;
st_mcAxis.rMaxAcceleration	:= 50000;
st_mcAxis.rMaxDeceleration	:= 50000;
st_mcAxis.rMaxJerk			:= 500000;
st_mcAxis.rAcceleration	:= 2500;
st_mcAxis.rDeceleration	:= 2500;
st_mcAxis.rJerk			:= 12500;
st_mcAxis.rMaxVelocity		:= 100;
st_mcAxis.rMaxDistance		:= 50;
st_mcAxis.bPosSen	:= TRUE ;//TODO link to digital input
st_mcAxis.bNegSen	:= TRUE ;//TODO link to digital input
st_mcAxis.mcHome.bCalibrationCam	:= TRUE;//TODO link to digital input origin
st_mcAxis.bPositionSensor	:= TRUE;//TODO link to digital input origin
st_mcAxis.bdirFW	:= TRUE;
st_mcAxis.sNetID := '192.168.11.159.5.1';
i	:= id_roller;
IF i=3 THEN
	st_mcAxis.nSlaveAddr	:= 1008;
END_IF

IF MAIN.firstCycle THEN
	st_mcAxis.mcPower.Enable	:= TRUE;
END_IF;
END_METHOD

METHOD M_reset : BOOL
VAR_INPUT
END_VAR
M_reset	:= FALSE;
ton_timeout.IN	:= FALSE;
eStates	:=E_RollerStates.IDLE;
xError	:= FALSE;
st_mcAxis.mcStop.Execute	:= FALSE;
st_mcAxis.mcReset.Execute	:= TRUE;
IF NOT roller.err THEN
	IF id_roller=3 THEN
		IF st_mcAxis.mcReadStatus.StandStill THEN
			M_reset	:= TRUE;
		END_IF
	ELSE
		M_reset	:= TRUE;		
	END_IF
END_IF
END_METHOD

METHOD M_safetyEvent : BOOL
VAR_INPUT
END_VAR
M_safetyEvent	:= FALSE;

roller.forward	:= FALSE;	
roller.backward	:= FALSE;
st_mcAxis.mcMoveAbsolute.Execute	:= FALSE;
st_mcAxis.mcStop.Execute	:= TRUE;

M_safetyEvent	:= TRUE;
END_METHOD

END_FUNCTION_BLOCK

// ---- Mian/machine/mcp/FB_mcp.TcPOU
FUNCTION_BLOCK FB_mcp
VAR_INPUT
	lightTower			: ST_LightTower;
END_VAR
VAR_OUTPUT
	
END_VAR
VAR_IN_OUT
	
END_VAR
VAR

	
	EDM_EES				: BOOL;
	EDM_EAS				: BOOL;
	st_safety_door		: ST_safetyDoor;
	st_control_pannel	: ST_control_pannel;
	
END_VAR

M_mapping();

METHOD M_mapping : BOOL
VAR_INPUT
END_VAR
/////////////////////////////////////digital input////////////////////////////////////////
st_control_pannel.button_start		:= G_IO.arDI[0].Ch[0];
st_control_pannel.button_stop		:= G_IO.arDI[0].Ch[1];
st_control_pannel.button_reset		:= G_IO.arDI[0].Ch[2];
st_control_pannel.button_power		:= G_IO.arDI[0].Ch[3];
EDM_EES								:= G_IO.arDI[0].Ch[4];
EDM_EAS								:= G_IO.arDI[0].Ch[5];
st_safety_door.button_reset			:= G_IO.arDI[0].Ch[6];
st_safety_door.button_unlock		:= G_IO.arDI[0].Ch[7];
st_safety_door.door_closed			:= G_IO.arDI[0].Ch[8];

/////////////////////////////////////digital output////////////////////////////////////////
G_IO.arDO[0].Ch[0]	:= st_control_pannel.lamp_start;
G_IO.arDO[0].Ch[1]	:= st_control_pannel.lamp_stop;
G_IO.arDO[0].Ch[2]	:= st_control_pannel.lamp_reset;
G_IO.arDO[0].Ch[3]	:= lightTower.RED;
G_IO.arDO[0].Ch[4]	:= lightTower.YELLOW;
G_IO.arDO[0].Ch[5]	:= lightTower.GREEN;
G_IO.arDO[0].Ch[6]	:= lightTower.BLUE;
G_IO.arDO[0].Ch[7]	:= lightTower.WHITE;
G_IO.arDO[0].Ch[8]	:= lightTower.BUZZER;
G_IO.arDO[0].Ch[9]	:= st_safety_door.lamp_reset;
G_IO.arDO[0].Ch[10]	:= st_safety_door.lamp_unlock;
G_IO.arDO[0].Ch[11]	:= st_safety_door.door_lock;
END_METHOD

END_FUNCTION_BLOCK

// ---- 02DUTs/Ads/FB_Tote_Subsystem.TcPOU
FUNCTION_BLOCK FB_Tote_Subsystem
VAR_INPUT
END_VAR
VAR_OUTPUT
END_VAR
VAR
	status	: MachineStatus := MachineStatus.STOPPED;
	workflow_status	: ToteSubsystemWorkflowStatus := ToteSubsystemWorkflowStatus.UNKNOWN;
	error_status	: OrderToteErrorStatus := OrderToteErrorStatus.UNKNOWN;
	loading_tote	: FB_ToteData;
	buffer_tote		: FB_ToteData;
	working_tote	: FB_ToteData;
	machine_control_cmd	: MachineControlCommand;
	autostore_control_cmd	: AutostoreControlCommand;
	autostore_status	: AutostoreStatus;

	cmd	: OrderToteCommand;
	iLoad	: INT;
	iUnload	: INT;
	ton1	: TON;
	working_tote_status	: ToteStatus;
	p_eTransfer_working	: POINTER TO E_Transfer;
///////////////////////////autostore mock////////////////	
	auto_store_run		: BOOL;
	auto_store_sensor	: BOOL;
	rtStop_auto_store	: R_TRIG;

END_VAR

M_mapping();
//status					:= GVL.machine_status;
workflow_status			:= GVL.fb_working.workflow_status;
error_status			:= GVL.fb_working.error_status;
working_tote._status	:= GVL.fb_working.tote_status;

p_eTransfer_working	:= ADR(GVL.fb_working.eTransfer);
CASE cmd OF
	OrderToteCommand.DO_NOTHING:
		p_eTransfer_working^ := E_Transfer.IDLE;
	OrderToteCommand.LOAD:
		IF GVL.fb_working.xUnloading THEN//avoid wrong command
			cmd	:= OrderToteCommand.DO_NOTHING;
			RETURN;
		END_IF
		p_eTransfer_working^ := E_Transfer.LOAD;
		IF GVL.fb_working.M_load() THEN
			cmd	:= OrderToteCommand.DO_NOTHING;
		END_IF			
	OrderToteCommand.OPEN_BAG:		
		;
	OrderToteCommand.STOP:
		;
	OrderToteCommand.SWAP:
		;
	OrderToteCommand.UNLOAD:
		IF GVL.fb_working.xLoading THEN//avoid wrong command
			cmd	:= OrderToteCommand.DO_NOTHING;
			RETURN;
		END_IF
		p_eTransfer_working^ := E_Transfer.UNLOAD;
		IF GVL.fb_working.M_unload() THEN
			cmd	:= OrderToteCommand.DO_NOTHING;
		END_IF
END_CASE


ton1(PT:=T#1S);

//////////////////////////mock autostore/////////////////
rtStop_auto_store(CLK:=auto_store_sensor);
IF MAIN.application.safety.xError THEN
	auto_store_run	:= FALSE;
	autostore_control_cmd	:= AutostoreControlCommand.DO_NOTHING;
END_IF
CASE autostore_control_cmd OF
	AutostoreControlCommand.DO_NOTHING:
		auto_store_run	:= FALSE;
	AutostoreControlCommand.START:
		auto_store_run	:= TRUE;
		autostore_status	:= AutostoreStatus.ROTATING;
		IF rtStop_auto_store.Q THEN
			auto_store_run	:= FALSE;
			autostore_status	:= AutostoreStatus.READY;
			autostore_control_cmd	:= AutostoreControlCommand.DO_NOTHING;
		END_IF
	AutostoreControlCommand.STOP:
		auto_store_run	:= FALSE;
		autostore_control_cmd	:= AutostoreControlCommand.DO_NOTHING;
END_CASE

{attribute 'TcRpcEnable'}
METHOD autostore_control_command : BOOL
VAR_INPUT
	Command	: AutostoreControlCommand;
END_VAR
autostore_control_command	:= FALSE; 
IF MAIN.eState=E_SystemManager.IN_PROGRESS AND autostore_control_cmd=AutostoreControlCommand.DO_NOTHING AND MAIN.application.safety.bStop_button_unlock THEN
	autostore_control_cmd	:= Command;
ELSE
	cmd	:= OrderToteCommand.DO_NOTHING;
END_IF
autostore_control_command	:= TRUE;
END_METHOD

METHOD M_Load : BOOL
VAR_INPUT
END_VAR
M_Load	:=FALSE;
CASE iLoad OF
	0:	
		working_tote._status	:= ToteStatus.EMPTY;
		workflow_status := ToteSubsystemWorkflowStatus.WAITING_FOR_NEW_TOTE;
		ton1.IN	:= FALSE;
		//GVL.iLoad	:= 1;
	1:
		ton1.IN	:= TRUE;
		IF ton1.Q THEN
			ton1.IN	:= FALSE;
			iLoad	:= 2;
		END_IF
	2:	
		workflow_status := ToteSubsystemWorkflowStatus.INBOUNDING;
		working_tote._status	:= ToteStatus.LOADED;
		iLoad	:= 3;
	3:
		ton1.IN	:= TRUE;
		IF ton1.Q THEN
			ton1.IN	:= FALSE;
			iLoad	:= 4;
		END_IF
	4:	
		workflow_status := ToteSubsystemWorkflowStatus.BAG_OPENING;
		working_tote._status	:= ToteStatus.READY;
		iLoad	:= 5;
	5:
		ton1.IN	:= TRUE;
		IF ton1.Q THEN
			ton1.IN	:= FALSE;
			iLoad	:= 6;
		END_IF		
	6:	
		workflow_status := ToteSubsystemWorkflowStatus.IDLE;
		iLoad	:= 0;
		M_Load	:= TRUE;
		GVL.fb_working.M_load();
END_CASE
END_METHOD

METHOD M_mapping : BOOL
VAR_INPUT
END_VAR
G_IO.arDO[0].Ch[13]	:= auto_store_run;
auto_store_sensor	:= G_IO.arDI[0].Ch[13];
END_METHOD

METHOD M_Swap : BOOL
VAR_INPUT
END_VAR
END_METHOD

METHOD M_Unload : BOOL
VAR_INPUT
END_VAR
M_Unload	:=FALSE;
CASE iUnload OF	
	0:	
		workflow_status := ToteSubsystemWorkflowStatus.WAITING_FOR_UNLOADING;
		ton1.IN	:= FALSE;
		iUnload	:= 1;
	1:
		ton1.IN	:= TRUE;
		IF ton1.Q THEN
			ton1.IN	:= FALSE;
			iUnload	:= 2;
		END_IF
	2:	
		workflow_status := ToteSubsystemWorkflowStatus.OUTBOUNDING;
		working_tote._status	:= ToteStatus.EMPTY;
		iUnload	:= 3;
	3:
		ton1.IN	:= TRUE;
		IF ton1.Q THEN
			ton1.IN	:= FALSE;
			iUnload	:= 4;
		END_IF	
	4:	
		workflow_status := ToteSubsystemWorkflowStatus.IDLE;
		iUnload	:= 0;
		M_Unload	:=TRUE;
END_CASE
END_METHOD

{attribute 'TcRpcEnable'}
METHOD machine_control_command : BOOL
VAR_INPUT
	Command	: MachineControlCommand;
END_VAR
machine_control_command	:= FALSE; 

machine_control_cmd	:= Command;

machine_control_command	:= TRUE;
END_METHOD

{attribute 'TcRpcEnable'}
METHOD order_tote_action_request : BOOL
VAR_INPUT
	Command	: OrderToteCommand;
END_VAR
order_tote_action_request	:= FALSE; 
IF MAIN.eState=E_SystemManager.IN_PROGRESS AND cmd=OrderToteCommand.DO_NOTHING AND MAIN.application.safety.bStop_button_unlock THEN
	cmd	:= Command;
ELSE
	error_status	:= OrderToteErrorStatus.MACHINE_NOT_RUNNING;
	cmd	:= OrderToteCommand.DO_NOTHING;
END_IF

order_tote_action_request	:= TRUE;
END_METHOD

END_FUNCTION_BLOCK

// ---- 02DUTs/Ads/FB_ToteData.TcPOU
FUNCTION_BLOCK FB_ToteData
VAR_INPUT
	
END_VAR
VAR_OUTPUT
END_VAR
VAR_IN_OUT
	
END_VAR
VAR
	status	: ToteStatus:= ToteStatus.UNKNOWN;
	barcode	: STRING	:= '';
	barcode_validation	: BarcodeVerificationResult	:= BarcodeVerificationResult.UNVERIFIED;
	
END_VAR

PROPERTY _status : ToteStatus
GET
_status	:= status;
END_GET
SET

status	:= _status;
END_SET
END_PROPERTY

END_FUNCTION_BLOCK

// ---- 02DUTs/Ads/FB_Light_tower_module.TcPOU
FUNCTION_BLOCK FB_Light_tower_module
VAR_INPUT
END_VAR
VAR_OUTPUT
END_VAR
VAR
	lightTower	: ST_LightTower;

END_VAR

IF MAIN.application.tote_subsystem.ton_heart_beat.Q THEN
	update_light_tower(0);
END_IF

PROPERTY _lightTower : ST_LightTower
GET
_lightTower	:= lightTower;
END_GET
SET
lightTower	:= _lightTower;
END_SET
END_PROPERTY

{attribute 'TcRpcEnable'}
METHOD update_light_tower : BOOL
VAR_INPUT
	iLightTowerStatus	: UINT;
END_VAR
update_light_tower	:= FALSE;
lightTower.GREEN	:= iLightTowerStatus.0;
lightTower.RED		:= iLightTowerStatus.1;
lightTower.WHITE	:= iLightTowerStatus.2;
lightTower.BLUE		:= iLightTowerStatus.3;
lightTower.YELLOW	:= iLightTowerStatus.4;
lightTower.BUZZER	:= iLightTowerStatus.5;
update_light_tower	:= TRUE;
END_METHOD

END_FUNCTION_BLOCK

// ---- Mian/statemachine/Prepare_Date_Time.TcPOU
FUNCTION Prepare_Date_Time : STRING(255)
VAR_INPUT
	str_DT									: Tc2_Utilities.TIMESTRUCT;
END_VAR
VAR
	tmp_str									: STRING(255);
	tmp_result								: STRING(255);
END_VAR

//fb_Time();

	tmp_result := Tc2_Standard.CONCAT('DATE ', WORD_TO_STRING(str_DT.wYear MOD 100));
	tmp_result := Tc2_Standard.CONCAT(tmp_result, '-');
	tmp_str    := WORD_TO_STRING(str_DT.wMonth);
	IF Tc2_Standard.LEN(tmp_str) < 2 THEN
		tmp_str := Tc2_Standard.CONCAT('0', tmp_str);
	END_IF;
	tmp_result := Tc2_Standard.CONCAT(tmp_result, tmp_str);
	
	tmp_result := Tc2_Standard.CONCAT(tmp_result, '-');
	tmp_str    := WORD_TO_STRING(str_DT.wDay);
	IF Tc2_Standard.LEN(tmp_str) < 2 THEN
		tmp_str := Tc2_Standard.CONCAT('0', tmp_str);
	END_IF;
	tmp_result := Tc2_Standard.CONCAT(tmp_result, tmp_str);

	tmp_result := Tc2_Standard.CONCAT(tmp_result, '  TIME ');
	tmp_str    := WORD_TO_STRING(str_DT.wHour);
	IF Tc2_Standard.LEN(tmp_str) < 2 THEN
		tmp_str := Tc2_Standard.CONCAT('0', tmp_str);
	END_IF;
	tmp_result := Tc2_Standard.CONCAT(tmp_result, tmp_str);

	tmp_result := Tc2_Standard.CONCAT(tmp_result, ':');
	tmp_str    := WORD_TO_STRING(str_DT.wMinute);
	IF Tc2_Standard.LEN(tmp_str) < 2 THEN
		tmp_str := Tc2_Standard.CONCAT('0', tmp_str);
	END_IF;
	tmp_result := Tc2_Standard.CONCAT(tmp_result, tmp_str);

	tmp_result := Tc2_Standard.CONCAT(tmp_result, ':');
	tmp_str    := WORD_TO_STRING(str_DT.wSecond);
	IF Tc2_Standard.LEN(tmp_str) < 2 THEN
		tmp_str := Tc2_Standard.CONCAT('0', tmp_str);
	END_IF;
	tmp_result := Tc2_Standard.CONCAT(tmp_result, tmp_str);
	
	tmp_result := Tc2_Standard.CONCAT(tmp_result, ':');
	tmp_str    := WORD_TO_STRING(str_DT.wMilliseconds);
	IF Tc2_Standard.LEN(tmp_str) = 1 THEN
		tmp_str := Tc2_Standard.CONCAT('00', tmp_str);
	END_IF;
	IF Tc2_Standard.LEN(tmp_str) = 2 THEN
		tmp_str := Tc2_Standard.CONCAT('0', tmp_str);
	END_IF;
	tmp_result := Tc2_Standard.CONCAT(tmp_result, tmp_str);	
	Prepare_Date_Time := tmp_result;

END_FUNCTION

// ---- Mian/Event_clear.TcPOU
FUNCTION Event_clear : BOOL
VAR_INPUT
END_VAR
VAR
	i: INT;
END_VAR

FOR i:=0 TO GVL.iAlarm_max DO
	GVL.events_alarm[i]	:= GVL.event_for_clear;
END_FOR

END_FUNCTION

// ---- GlobalTextList.TcGTLO
TEXTLIST GlobalTextList
  206 = '%.2f mm'
  740 = '%.3f mm'
  201 = '%s'
  209 = '+'
  210 = '-'
  602 = 'Acc'
  843 = 'Actual Position'
  773 = 'Aging test'
  5 = 'Alarm'
  203 = 'Axis Error '
  299 = 'Axis_bagOpen_0'
  618 = 'Axis_bagOpen_1'
  211 = 'Axis_bagOpen_2'
  743 = 'Axis_bagOpen_3'
  324 = 'Axis_vacuun_0'
  786 = 'Axis_vacuun_1'
  179 = 'BagOpen'
  81 = 'BELT ESTOP'
  808 = 'Breaker OFF'
  486 = 'Breaker ON'
  1159 = 'buffer'
  327 = 'BUFFER SAFETY'
  732 = 'Buffer Stopper'
  349 = 'Dec'
  216 = 'deg/s'
  217 = 'deg/s²'
  180 = 'DIO'
  662 = 'DOG'
  673 = 'error'
  924 = 'Extend'
  614 = 'extended'
  801 = 'Flood Light'
  841 = 'HOME'
  248 = 'HomeDone'
  902 = 'ID'
  136 = 'inbound'
  44 = 'INIT'
  708 = 'Message'
  361 = 'Method'
  737 = 'name'
  1029 = 'outbound_end'
  706 = 'photo_sens[1]or_start'
  681 = 'sensor_start[0]'
  1006 = 'sensor_start[1]'
  102 = 'sStepID'
  99 = 'Jerk'
  839 = 'JOG BW'
  840 = 'JOG FW'
  1374 = 'lift'
  795 = 'LIFT'
  178 = 'Lift'
  926 = 'LIFT ESTOP'
  519 = 'LIFT STATION DETECTION'
  495 = 'LIGHT CURTAIN LEFT'
  39 = 'LIGHT CURTAIN RIGHT'
  413 = 'LOAD'
  897 = 'LOADING SAFETY'
  351 = 'Main'
  386 = 'MCP ESTOP'
  215 = 'mm/s'
  214 = 'mm/s²'
  207 = 'MOVE ABS'
  569 = 'Move relative'
  205 = 'Neg LS'
  677 = 'outbound'
  842 = 'photosensor[0]'
  79 = 'photosensor[1]'
  70 = 'photo_sensor[0]'
  919 = 'photo_sensor[1]'
  800 = 'photo_sensor_mute'
  925 = 'photo_sensor_mute_l'
  891 = 'photo_sensor_start'
  1003 = 'place'
  204 = 'Pos LS'
  844 = 'Power \nOn'
  359 = 'Power On'
  342 = 'ReM'
  1185 = 'ReM3'
  904 = 'ReM4'
  274 = 'ReM5'
  199 = 'Reset'
  10 = 'RESET'
  1651 = 'retract'
  934 = 'retracted'
  71 = 'ROBOT EAS'
  312 = 'ROBOT EES'
  72 = 'roller'
  1437 = 'Roller In'
  189 = 'roller[0]'
  709 = 'roller[1]'
  633 = 'roller[2]'
  687 = 'roller[3]'
  522 = 'roller_x'
  792 = 'roller_y'
  845 = 'RUN'
  634 = 'SAFETY DOOR'
  202 = 'SAFETY INPUT'
  617 = 'SAFETY OUTPUT'
  641 = 'sComponentID'
  438 = 'sComponent_ID'
  358 = 'sComponent_name'
  874 = 'sensor_mute'
  143 = 'sensor_mute_left'
  487 = 'sensor_mute_right'
  622 = 'Set absolute\nencoder as linear'
  454 = 'Set absolute\nencoder as rotation'
  208 = 'Set Point'
  14 = 'Set Pos to 0'
  332 = 'sEventType'
  714 = 'sEvent_MSG'
  245 = 'sID'
  220 = 'sMethod'
  1034 = 'StepID'
  986 = 'sTime'
  198 = 'Stop'
  996 = 'STOP'
  666 = 'Time'
  784 = 'tote_detection'
  585 = 'Type'
  780 = 'UNLOAD'
  863 = 'valve_clamp[0]'
  396 = 'valve_lift'
  464 = 'valve_lift[0]'
  227 = 'valve_stopper'
  200 = 'Velocity'
  193 = 'WORKING SAFETY'
END_TEXTLIST

// ---- VISUs/VISUs/Menu.TcVIS
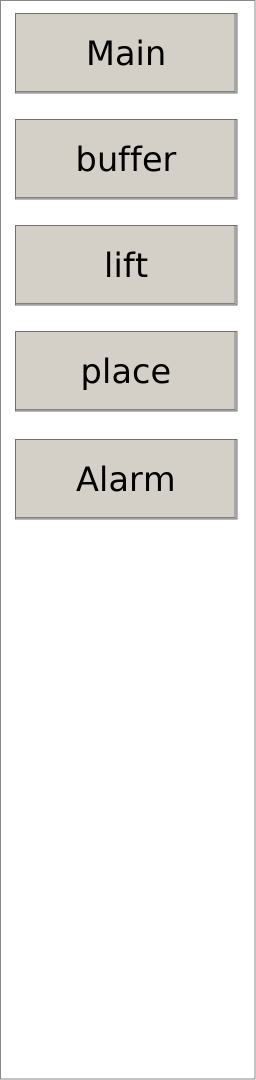
VISUALIZATION Menu  // 256x1080
    Button (15,119 222x80), "buffer", colour toggle: G_HMI.iMainFrame =1
        p573394764: 16#FF00FF00
        OnMouseDown: execute { G_HMI.iMainFrame	:= 1; }
    Button (15,225 222x80), "lift", colour toggle: G_HMI.iMainFrame =2
        p573394764: 16#FF00FF00
        OnMouseDown: execute { G_HMI.iMainFrame	:= 2; }
    Button (15,331 222x80), "place", colour toggle: G_HMI.iMainFrame =3
        p573394764: 16#FF00FF00
        OnMouseDown: execute { G_HMI.iMainFrame	:= 3; }
    Button (15,13 222x80), "Main", colour toggle: G_HMI.iMainFrame =0
        p573394764: 16#FF00FF00
        OnMouseDown: execute { G_HMI.iMainFrame	:= 0; }
    Button (15,439 222x80), "Alarm", colour toggle: G_HMI.iMainFrame =4
        p573394764: 16#FF00FF00
        OnMouseDown: execute { G_HMI.iMainFrame	:= 4; }
END_VISUALIZATION

// ---- VISUs/VISUs/visu_buffer.TcVIS
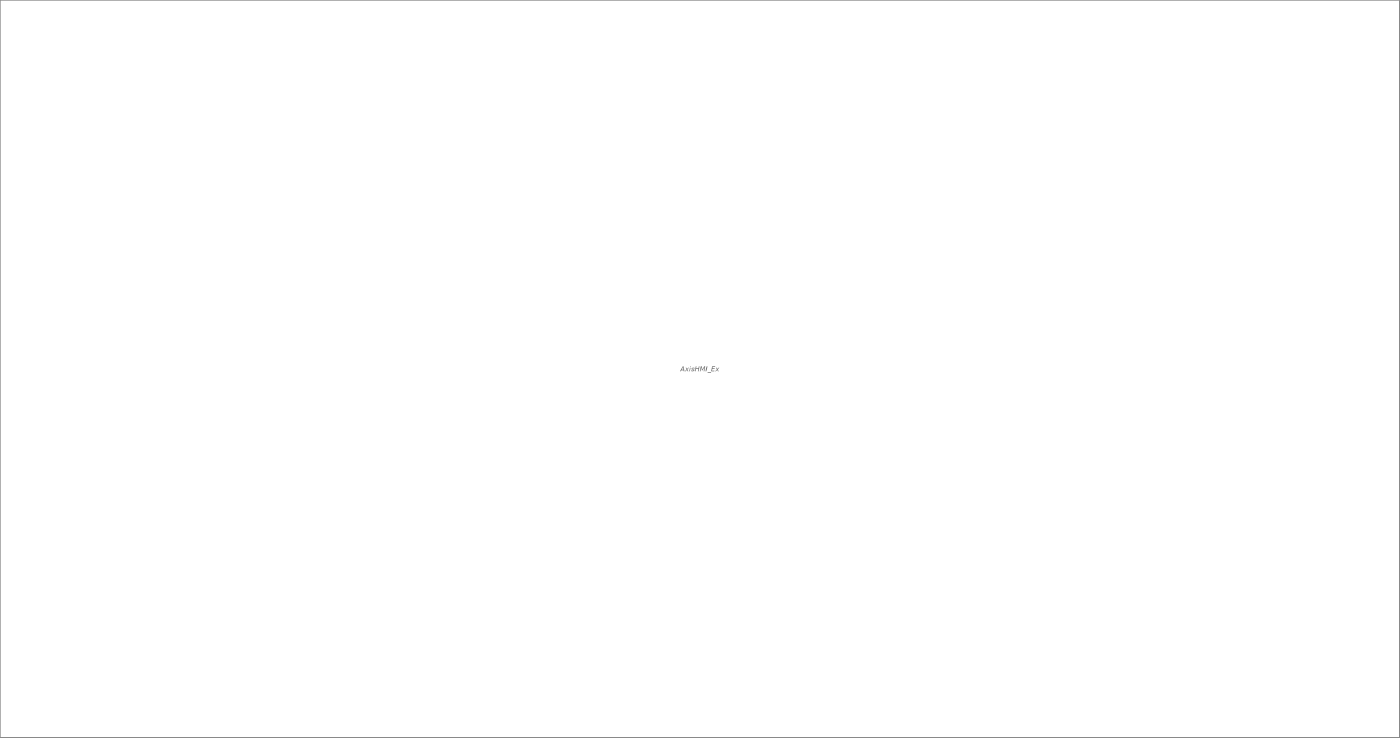
VISUALIZATION visu_buffer  // 2048x1080
    TabControl (0,0 2048x1080)
        shows AxisHMI_Ex(stAxisHMI := GVL.fb_buffer.fb_rollers[3].st_mcAxis, mcAxis := GVL.fb_buffer.fb_rollers[3].mcAxis, xError := GVL.fb_buffer.fb_rollers[3].mcAxis.xError)
        shows v_io_buffer()
        shows Axis_HMI(st_axis_HMI := st_mcAxis[EN_Axis.Grip_axis])
        shows AxisMotionLib.AxisHMI_Ex(stAxisHMI := gantrybase.st_mcAxis[EN_Axis.Z], mcAxis := gantrybase.mcAxis[EN_Axis.Z], xError := gantrybase.mcAxis[EN_Axis.Z].xError)
        shows v_rem_1(dIO_ReM := GVL.rem[G_HMI.iReM])
        [0]: TabTitle=Buffer Stopper
        [6]: TabTitle=Gripper
        [1]: AxisHMI=gantrybase.st_mcAxis[EN_Axis.Y], mcAxis=gantrybase.mcAxis[EN_Axis.Y], Error=gantrybase.mcAxis[EN_Axis.Y].xError
        [3]: TabTitle=ReMIO_1
        p699000190: gantrybase.st_mcAxis[EN_Axis.X]
        p2837713833: gantrybase.mcAxis[EN_Axis.Z].sAxisName
        p520277221: gantrybase.mcAxis[EN_Axis.X].xError
        p3331604638: gantrybase.st_mcAxis[EN_Axis.Z]
        p1813558639: gantrybase.mcAxis[EN_Axis.Z].xError
        p1563495665: gantrybase.st_mcAxis[EN_Axis.Y]
        p2070126892: gantrybase.mcAxis[EN_Axis.Y].xError
        p3435970784: gantrybase.mcAxis[EN_Axis.X]
        p2829954345: gantrybase.mcAxis[EN_Axis.Y]
        p3218520426: gantrybase.mcAxis[EN_Axis.Z]
END_VISUALIZATION

// ---- VISUs/VISUs/visu_loading.TcVIS
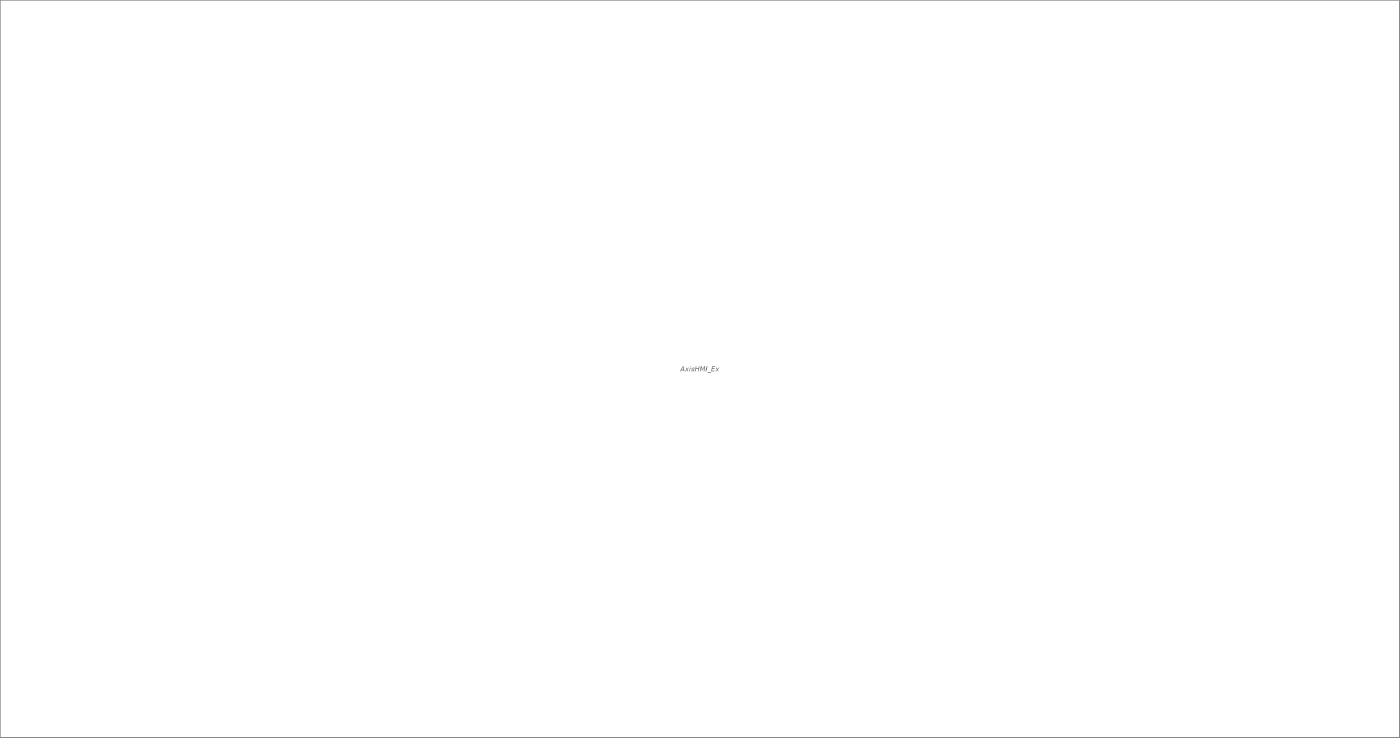
VISUALIZATION visu_loading  // 2048x1080
    TabControl (0,0 2048x1080)
        shows AxisHMI_Ex(stAxisHMI := GVL.FB_loading.st_mcAxis, mcAxis := GVL.FB_loading.mcAxis, xError := GVL.FB_loading.mcAxis.xError)
        shows v_io_loading()
        shows Axis_HMI(st_axis_HMI := st_mcAxis[EN_Axis.Grip_axis])
        shows v_placeModule_io()
        shows v_rem_1(dIO_ReM := GVL.rem[G_HMI.iReM])
        [0]: TabTitle=Lift
        [6]: TabTitle=Gripper
        [1]: AxisHMI=gantrybase.st_mcAxis[EN_Axis.Y], mcAxis=gantrybase.mcAxis[EN_Axis.Y], Error=gantrybase.mcAxis[EN_Axis.Y].xError
        [2]: AxisHMI=gantrybase.st_mcAxis[EN_Axis.Z], mcAxis=gantrybase.mcAxis[EN_Axis.Z], Error=gantrybase.mcAxis[EN_Axis.Z].xError
        [3]: TabTitle=ReMIO_1
        p699000190: gantrybase.st_mcAxis[EN_Axis.X]
        p2837713833: gantrybase.mcAxis[EN_Axis.Z].sAxisName
        p520277221: gantrybase.mcAxis[EN_Axis.X].xError
        p3331604638: gantrybase.st_mcAxis[EN_Axis.Z]
        p1813558639: gantrybase.mcAxis[EN_Axis.Z].xError
        p1563495665: gantrybase.st_mcAxis[EN_Axis.Y]
        p2070126892: gantrybase.mcAxis[EN_Axis.Y].xError
        p3435970784: gantrybase.mcAxis[EN_Axis.X]
        p2829954345: gantrybase.mcAxis[EN_Axis.Y]
        p3218520426: gantrybase.mcAxis[EN_Axis.Z]
END_VISUALIZATION

// ---- VISUs/VISUs/visu_main.TcVIS
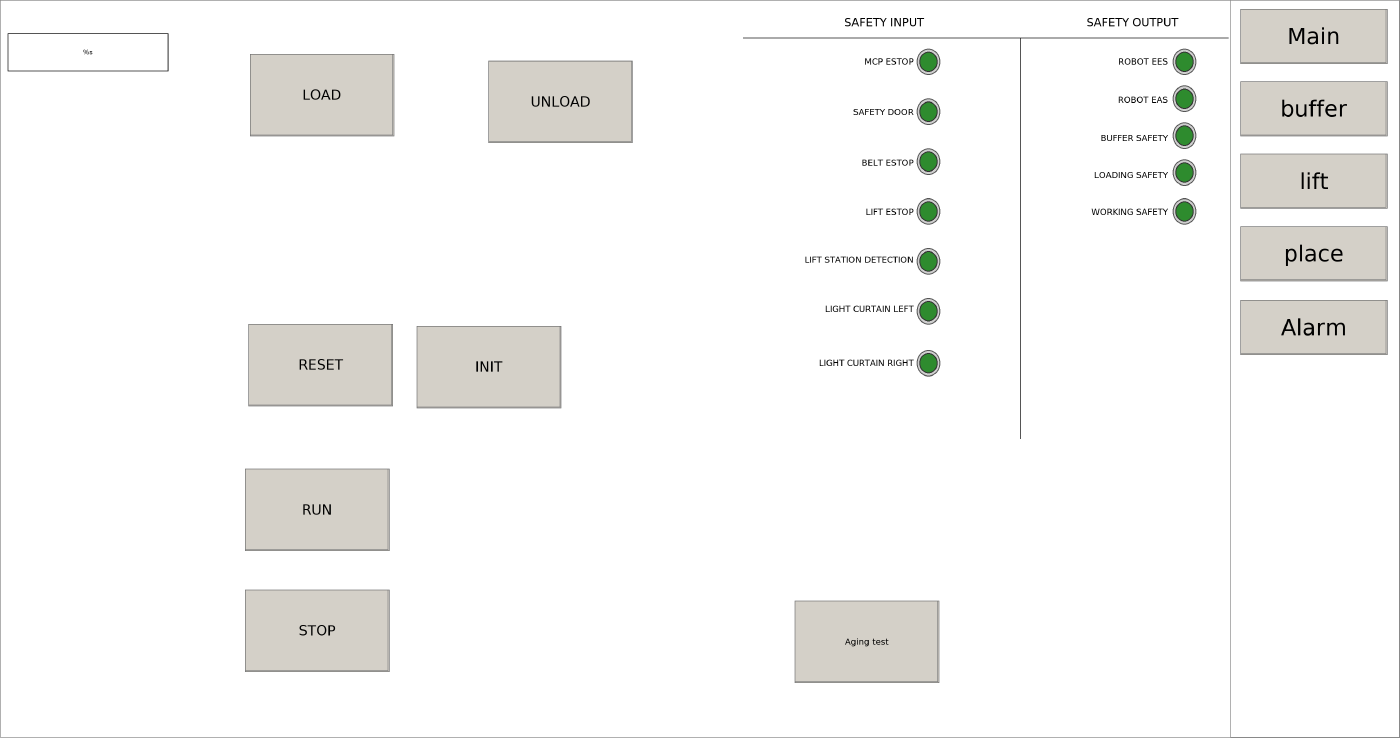
VISUALIZATION visu_main  // 2048x1080
    Frame (0,0 1800x1080), frame switch variable: G_HMI.iMainFrame
        shows visu_operation()
        shows visu_buffer()
        shows visu_loading()
        shows visu_working()
        shows v_alarm()
        shows v_IO_fixtureClamp()
    Frame (1800,0 248x1080), frame switch variable: G_HMI.iMainFrame
        shows Menu()
        shows visu_working()
        shows v_IO_fixtureClamp()
        shows visu_buffer()
        shows visu_loading()
        shows v_alarm()
END_VISUALIZATION

// ---- VISUs/VISUs/visu_operation.TcVIS
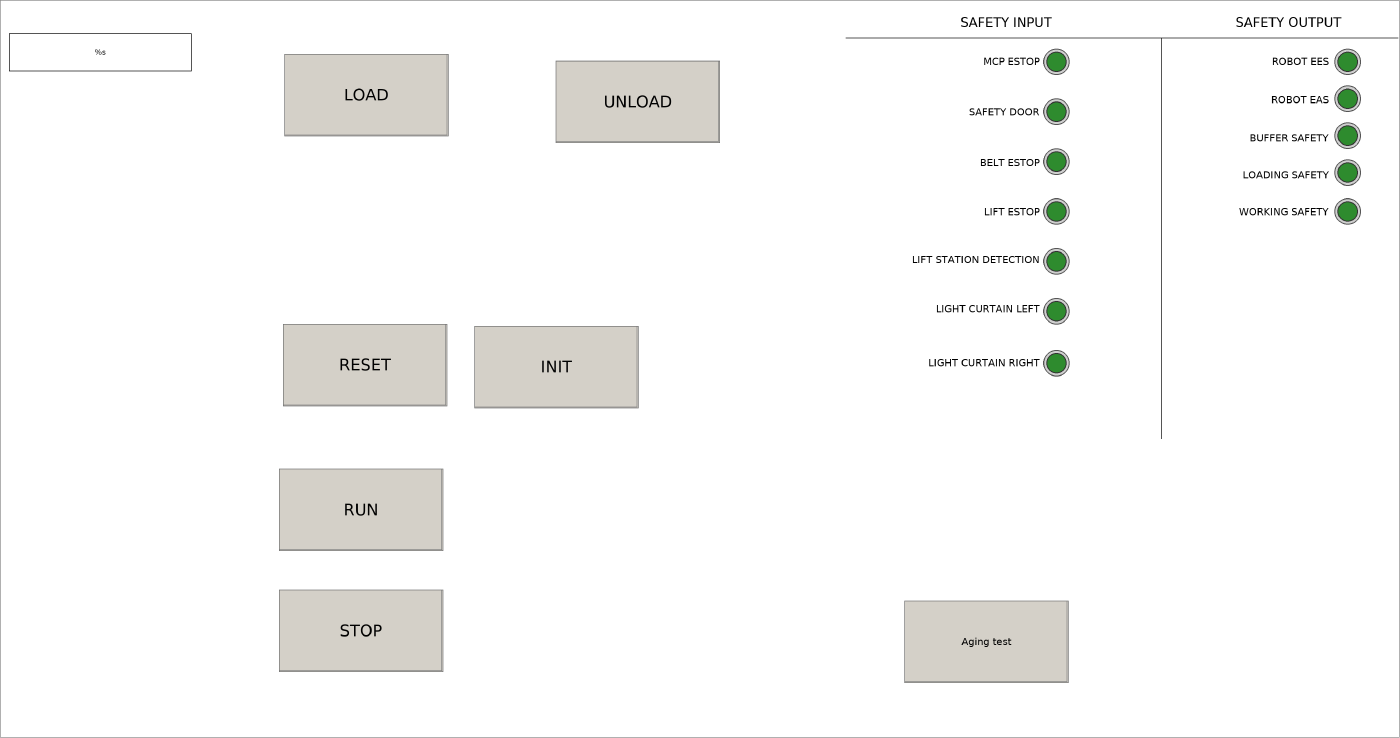
VISUALIZATION visu_operation  // 2048x1080
    Button (414,474 240x120), "RESET", colour toggle: G_HMI.bReset
        OnMouseDown: execute { G_HMI.bReset	:= TRUE; }
        OnMouseUp: execute { G_HMI.bReset	:= FALSE; }
    Button (408,686 240x120), "RUN", colour toggle: GVL.bRunning
        OnMouseDown: execute { G_HMI.bRun	:= TRUE; }
        OnMouseUp: execute { G_HMI.bRun	:= FALSE; }
    Button (694,477 240x120), "INIT", colour toggle: G_HMI.bInit
        OnMouseDown: execute { G_HMI.bInit	:= TRUE; }
        OnMouseUp: execute { G_HMI.bInit	:= FALSE; }
    Lamp1 (1523,68 45x45), variable: MAIN.application.safety.mcp_estop, style: Lamp-Lamp1-Green
    Label (1274,75 250x30), "MCP ESTOP"
    Lamp1 (1523,214 45x45), variable: MAIN.application.safety.belt_estop, style: Lamp-Lamp1-Green
    Label (1274,223 250x30), "BELT ESTOP"
    Lamp1 (1523,287 45x45), variable: MAIN.application.safety.lift_estop, style: Lamp-Lamp1-Green
    Label (1274,297 250x26), "LIFT ESTOP"
    Lamp1 (1523,360 45x45), variable: MAIN.application.safety.lift_station_detection, style: Lamp-Lamp1-Green
    Label (1274,367 250x26), "LIFT STATION DETECTION"
    Lamp1 (1523,141 45x45), variable: MAIN.application.safety.mcp_safetyDoor, style: Lamp-Lamp1-Green
    Label (1274,149 250x30), "SAFETY DOOR"
    Lamp1 (1523,433 45x45), variable: MAIN.application.safety.lift_lightCurtain_left, style: Lamp-Lamp1-Green
    Label (1274,437 250x30), "LIGHT CURTAIN LEFT"
    Lamp1 (1523,509 45x45), variable: MAIN.application.safety.lift_lightCurtain_right, style: Lamp-Lamp1-Green
    Label (1274,516 250x30), "LIGHT CURTAIN RIGHT"
    Lamp1 (1949,68 45x45), variable: MAIN.application.safety.robot_EES, style: Lamp-Lamp1-Green
    Label (1697,75 250x30), "ROBOT EES"
    Lamp1 (1949,176 45x45), variable: MAIN.application.safety.buffer_safety, style: Lamp-Lamp1-Green
    Label (1697,187 250x30), "BUFFER SAFETY"
    Lamp1 (1949,230 45x45), variable: MAIN.application.safety.loading_safety, style: Lamp-Lamp1-Green
    Label (1697,243 250x26), "LOADING SAFETY"
    Lamp1 (1949,287 45x45), variable: MAIN.application.safety.working_safety, style: Lamp-Lamp1-Green
    Label (1697,297 250x26), "WORKING SAFETY"
    Lamp1 (1949,122 45x45), variable: MAIN.application.safety.robot_EAS, style: Lamp-Lamp1-Green
    Label (1697,131 250x30), "ROBOT EAS"
    Line (1699,642) (1699,55)
    Label (1347,18 250x30), "SAFETY INPUT"
    Label (1760,18 250x30), "SAFETY OUTPUT"
    Line (1237,55) (2045,55)
    Button (416,79 240x120), "LOAD", invisible if: MAIN.application.tote_subsystem.cmd<>OrderToteCommand.DO_NOTHING, input disabled if: MAIN.application.tote_subsystem.cmd<>OrderToteCommand.DO_NOTHING
        OnMouseDown: execute { MAIN.application.tote_subsystem.cmd	:= OrderToteCommand.LOAD; }
        OnMouseUp: execute {  }
    Button (813,89 240x120), "UNLOAD", invisible if: MAIN.application.tote_subsystem.cmd<>OrderToteCommand.DO_NOTHING, input disabled if: MAIN.application.tote_subsystem.cmd<>OrderToteCommand.DO_NOTHING
        OnMouseDown: execute { MAIN.application.tote_subsystem.cmd	:= OrderToteCommand.UNLOAD; }
        OnMouseUp: execute {  }
    Button (1323,879 240x120), "Aging test", colour toggle: G_HMI.bAging_test
        OnMouseDown: execute { G_HMI.bAging_test	:= TRUE; }
        OnMouseUp: execute { G_HMI.bAging_test	:= FALSE; }
    Button (408,863 240x120), "STOP", colour toggle: GVL.bAck_stop
        OnMouseDown: execute { G_HMI.bStop	:= TRUE; }
        OnMouseUp: execute { G_HMI.bStop	:= FALSE; }
    Rectangle (13,49 267x55), "%s", text variable: MAIN.str_state
END_VISUALIZATION

// ---- VISUs/VISUs/visu_working.TcVIS
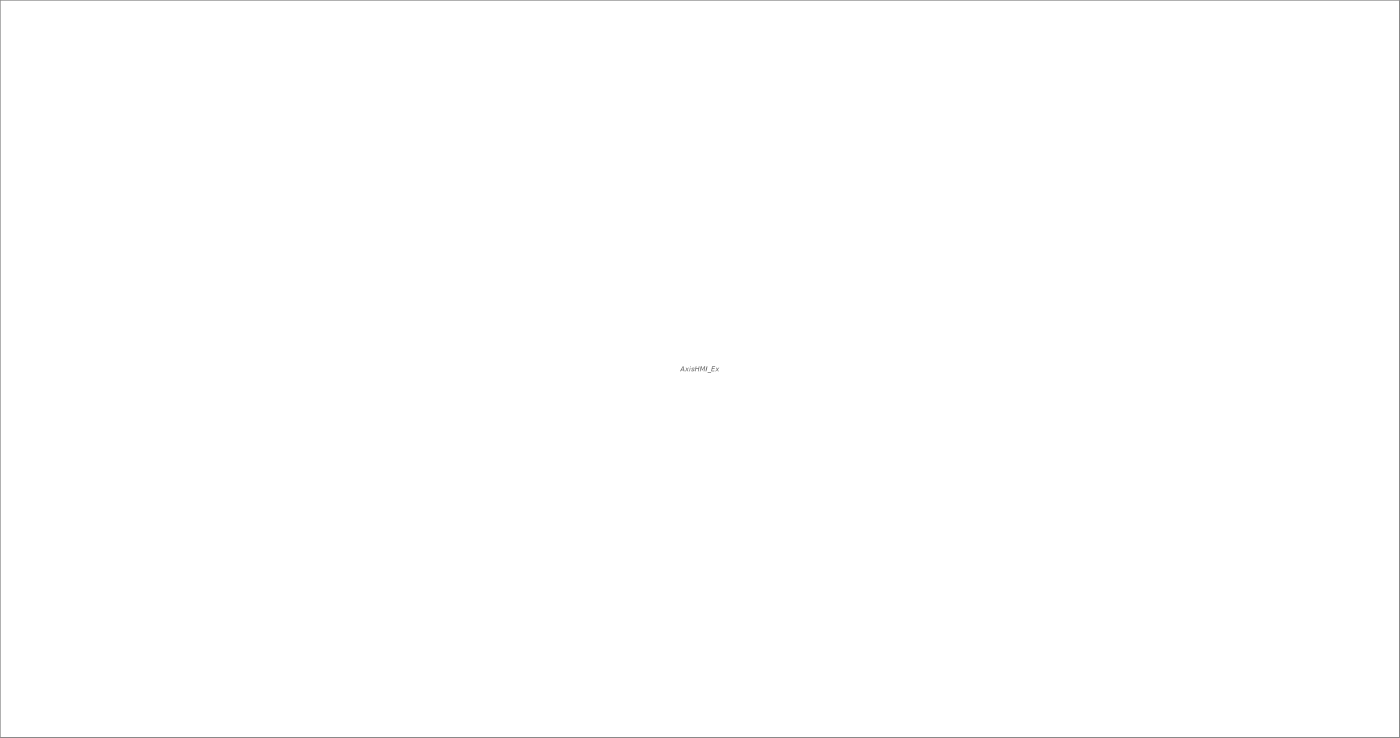
VISUALIZATION visu_working  // 2048x1080
    TabControl (0,0 2048x1080)
        shows AxisHMI_Ex(stAxisHMI := GVL.fb_working.st_mcAxis_lift, mcAxis := GVL.fb_working.mcAxis_lift, xError := GVL.fb_working.mcAxis_lift.xError)
        shows AxisHMI_Ex(stAxisHMI := GVL.fb_working.st_mcAxis_bag, mcAxis := GVL.fb_working.mcAxis_bag, xError := GVL.fb_working.mcAxis_bag.xError)
        shows v_io_working()
        shows AxisHMI_Ex(stAxisHMI := GVL.fb_working.st_mcAxis_vacuun[0], mcAxis := GVL.fb_working.mcAxis_vacuun[0], xError := GVL.fb_working.mcAxis_vacuun[0].xError)
        shows AxisHMI_Ex(stAxisHMI := GVL.fb_working.st_mcAxis_vacuun[1], mcAxis := GVL.fb_working.mcAxis_vacuun[1], xError := GVL.fb_working.mcAxis_vacuun[1].xError)
        shows AxisHMI_Ex(stAxisHMI := GVL.fb_working.st_mcAxis_bagOpen[0], mcAxis := GVL.fb_working.mcAxis_bagOpen[0], xError := GVL.fb_working.mcAxis_bagOpen[0].xError)
        shows AxisHMI_Ex(stAxisHMI := GVL.fb_working.st_mcAxis_bagOpen[1], mcAxis := GVL.fb_working.mcAxis_bagOpen[1], xError := GVL.fb_working.mcAxis_bagOpen[1].xError)
        shows AxisHMI_Ex(stAxisHMI := GVL.fb_working.st_mcAxis_bagOpen[2], mcAxis := GVL.fb_working.mcAxis_bagOpen[2], xError := GVL.fb_working.mcAxis_bagOpen[2].xError)
        shows AxisHMI_Ex(stAxisHMI := GVL.fb_working.st_mcAxis_bagOpen[3], mcAxis := GVL.fb_working.mcAxis_bagOpen[3], xError := GVL.fb_working.mcAxis_bagOpen[3].xError)
        [0]: TabTitle=Lift
        [1]: TabTitle=BagOpen
        [3]: TabTitle=Axis_vacuun_0
        [4]: TabTitle=Axis_vacuun_1
        [5]: TabTitle=Axis_bagOpen_0
        [6]: TabTitle=Axis_bagOpen_1
        [7]: TabTitle=Axis_bagOpen_2
        [8]: TabTitle=Axis_bagOpen_3
        p2837713833: gantrybase.mcAxis[EN_Axis.Z].sAxisName
END_VISUALIZATION

// ---- VISUs/VISUs/v_io_buffer.TcVIS
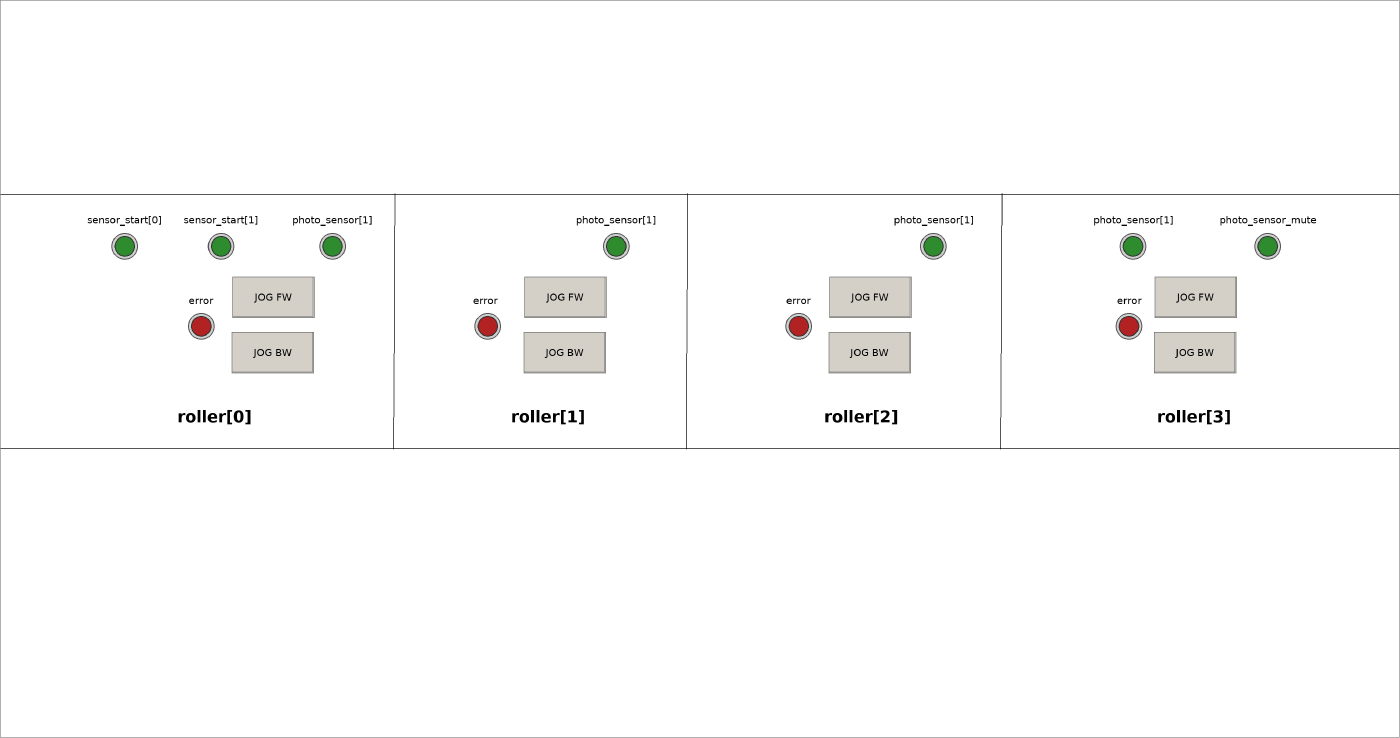
VISUALIZATION v_io_buffer  // 2048x1080
    Lamp1 (464,338 45x45), variable: GVL.fb_buffer.fb_rollers[0].roller.sensor.Q, style: Lamp-Lamp1-Green
    Label (386,309 200x26), "photo_sensor[1]"
    Lamp1 (272,455 45x45), variable: GVL.fb_buffer.fb_rollers[0].roller.err, style: Lamp-Lamp1-Red
    Label (194,427 200x26), "error"
    Label (248,597 132x26), "roller[0]"
    Line (0,284) (2048,284)
    Button (340,405 120x60), "JOG FW", colour toggle: GVL.fb_buffer.fb_rollers[0].roller.forward
        OnMouseDown: execute { GVL.fb_buffer.fb_rollers[0].roller.forward	:= TRUE; }
        OnMouseUp: execute { GVL.fb_buffer.fb_rollers[0].roller.forward	:= FALSE; }
    Button (339,486 120x60), "JOG BW", colour toggle: GVL.fb_buffer.fb_rollers[0].roller.backward
        OnMouseDown: execute { GVL.fb_buffer.fb_rollers[0].roller.backward	:= TRUE; }
        OnMouseUp: execute { GVL.fb_buffer.fb_rollers[0].roller.backward	:= FALSE; }
    Line (0,656) (2048,656)
    Lamp1 (160,338 45x45), variable: GVL.fb_buffer.sensor_start[0].Q, style: Lamp-Lamp1-Green
    Label (82,309 200x26), "sensor_start[0]"
    Lamp1 (879,338 45x45), variable: GVL.fb_buffer.fb_rollers[1].roller.sensor.Q, style: Lamp-Lamp1-Green
    Label (801,309 200x26), "photo_sensor[1]"
    Lamp1 (691,455 45x45), variable: GVL.fb_buffer.fb_rollers[1].roller.err, style: Lamp-Lamp1-Red
    Label (610,427 200x26), "error"
    Label (736,597 132x26), "roller[1]"
    Button (767,405 120x60), "JOG FW", colour toggle: GVL.fb_buffer.fb_rollers[1].roller.forward
        OnMouseDown: execute { GVL.fb_buffer.fb_rollers[1].roller.forward	:= TRUE; }
        OnMouseUp: execute { GVL.fb_buffer.fb_rollers[1].roller.forward	:= FALSE; }
    Button (766,486 120x60), "JOG BW", colour toggle: GVL.fb_buffer.fb_rollers[1].roller.backward
        OnMouseDown: execute { GVL.fb_buffer.fb_rollers[1].roller.backward	:= TRUE; }
        OnMouseUp: execute { GVL.fb_buffer.fb_rollers[1].roller.backward	:= FALSE; }
    Lamp1 (1343,338 45x45), variable: GVL.fb_buffer.fb_rollers[2].roller.sensor.Q, style: Lamp-Lamp1-Green
    Label (1266,309 200x26), "photo_sensor[1]"
    Lamp1 (1146,455 45x45), variable: GVL.fb_buffer.fb_rollers[2].roller.err, style: Lamp-Lamp1-Red
    Label (2867,952 200x26), "error"
    Label (1194,597 132x26), "roller[2]"
    Button (1213,405 120x60), "JOG FW", colour toggle: GVL.fb_buffer.fb_rollers[2].roller.forward
        OnMouseDown: execute { GVL.fb_buffer.fb_rollers[2].roller.forward	:= TRUE; }
        OnMouseUp: execute { GVL.fb_buffer.fb_rollers[2].roller.forward	:= FALSE; }
    Button (1212,486 120x60), "JOG BW", colour toggle: GVL.fb_buffer.fb_rollers[2].roller.backward
        OnMouseDown: execute { GVL.fb_buffer.fb_rollers[2].roller.backward	:= TRUE; }
        OnMouseUp: execute { GVL.fb_buffer.fb_rollers[2].roller.backward	:= FALSE; }
    Lamp1 (1635,338 45x45), variable: GVL.fb_buffer.fb_rollers[3].roller.sensor.Q, style: Lamp-Lamp1-Green
    Label (1558,309 200x26), "photo_sensor[1]"
    Lamp1 (1629,455 45x45), variable: GVL.fb_buffer.fb_rollers[2].roller.err, style: Lamp-Lamp1-Red
    Label (1552,427 200x26), "error"
    Label (1681,597 132x26), "roller[3]"
    Button (1689,405 120x60), "JOG FW", colour toggle: GVL.fb_buffer.fb_rollers[3].roller.forward
        OnMouseDown: execute { GVL.fb_buffer.fb_rollers[3].roller.forward	:= TRUE; }
        OnMouseUp: execute { GVL.fb_buffer.fb_rollers[3].roller.forward	:= FALSE; }
    Button (1688,486 120x60), "JOG BW", colour toggle: GVL.fb_buffer.fb_rollers[3].roller.backward
        OnMouseDown: execute { GVL.fb_buffer.fb_rollers[3].roller.backward	:= TRUE; }
        OnMouseUp: execute { GVL.fb_buffer.fb_rollers[3].roller.backward	:= FALSE; }
    Lamp1 (1832,338 45x45), variable: GVL.fb_buffer.fb_rollers[3].sensor_mute.Q, style: Lamp-Lamp1-Green
    Label (1755,309 200x26), "photo_sensor_mute"
    Lamp1 (301,338 45x45), variable: GVL.fb_buffer.sensor_start[1].Q, style: Lamp-Lamp1-Green
    Label (223,309 200x26), "sensor_start[1]"
    Line (576,657) (578,283)
    Line (1004,657) (1006,283)
    Line (1464,657) (1466,283)
    Label (1068,427 200x26), "error"
END_VISUALIZATION

// ---- VISUs/VISUs/v_alarm.TcVIS
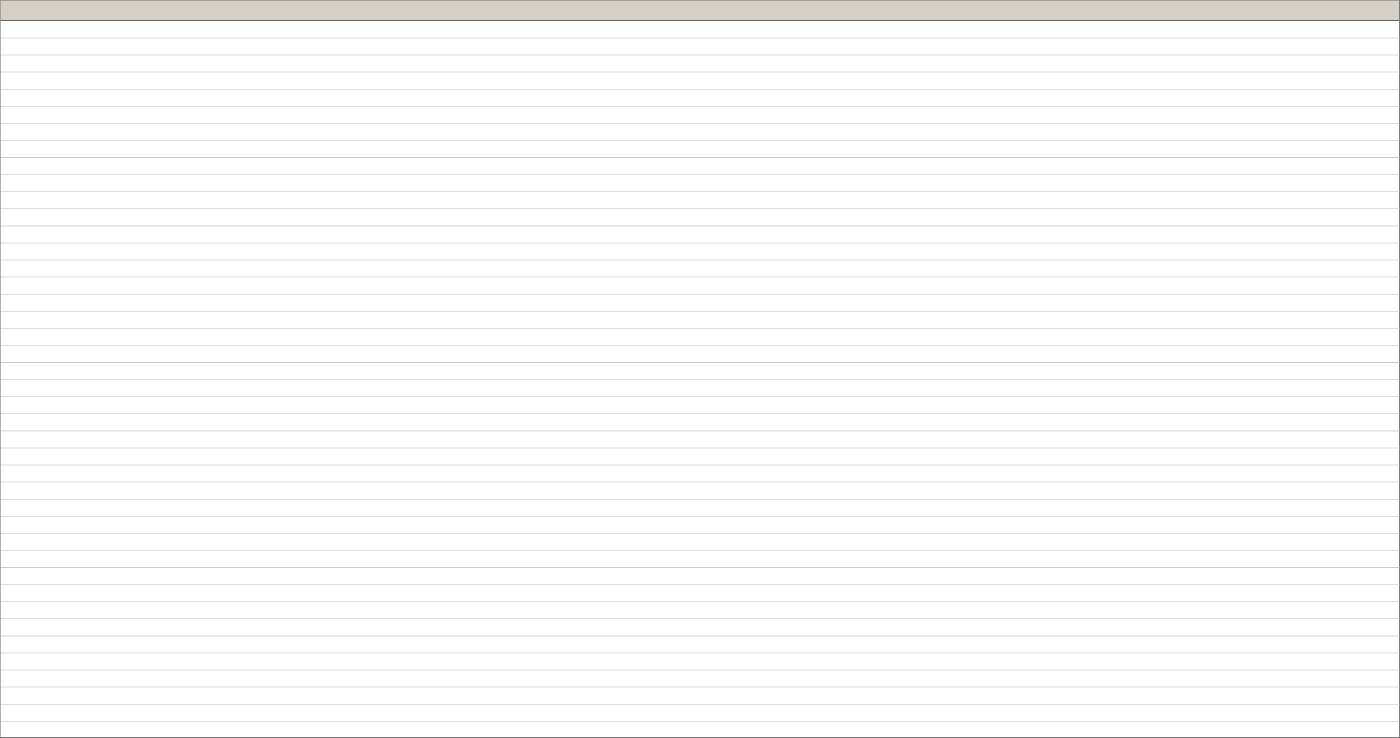
VISUALIZATION v_alarm  // 2048x1080
    Table (0,0 2048x1080), data array: GVL.events_alarm
        p3104783080: GVL.fb_buffer.fb_rollers[INDEX].AxisRef
        p2501879983: GVL.fb_buffer.fb_rollers[INDEX].current_tote_status
        p7306298: GVL.fb_buffer.fb_rollers[INDEX].ton_timeout
        p1933151965: GVL.fb_buffer.fb_rollers[INDEX].eStates
        p3863566920: GVL.fb_buffer.fb_rollers[INDEX].iStateTemp
        p2192122294: GVL.fb_buffer.fb_rollers[INDEX].errorMessage
        p400160035: GVL.fb_buffer.fb_rollers[INDEX].xError
        p1265227338: GVL.fb_buffer.fb_rollers[INDEX].rPos_up
        p3726181087: GVL.fb_buffer.fb_rollers[INDEX].rPos_down
        p3854506369: GVL.events_alarm[INDEX].sTime
        p1892666644: GVL.events_alarm[INDEX].sEventType
        p338671338: GVL.events_alarm[INDEX].sComponent_name
        p2170511999: GVL.events_alarm[INDEX].sComponentID
        p3723444502: GVL.events_alarm[INDEX].sMethod
        p1218418051: GVL.events_alarm[INDEX].sStepID
        p746581629: GVL.events_alarm[INDEX].sEvent_MSG
END_VISUALIZATION

// ---- VISUs/VISUs/v_io_loading.TcVIS
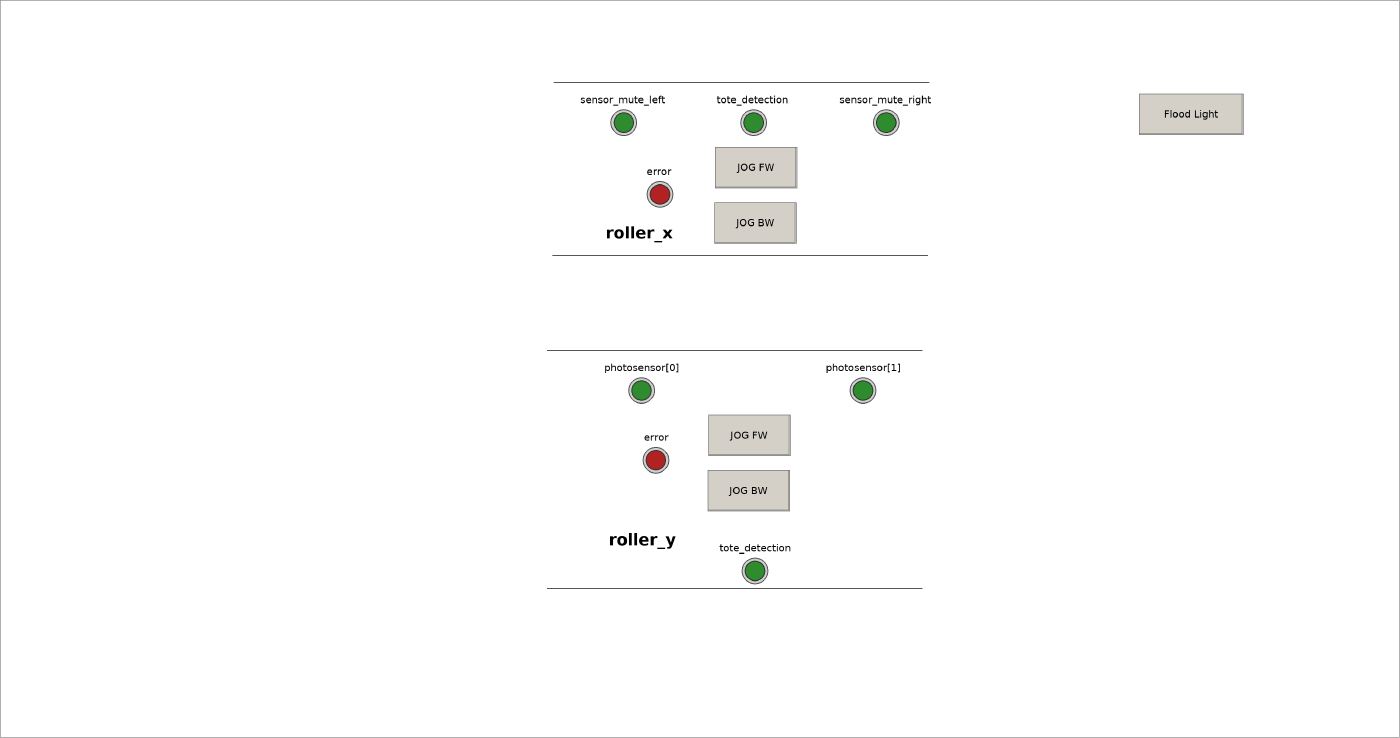
VISUALIZATION v_io_loading  // 2048x1080
    Lamp1 (1080,157 45x45), variable: GVL.fb_loading.photo_sensor_tote_detection.Q, style: Lamp-Lamp1-Green
    Label (1001,133 200x26), "tote_detection"
    Lamp1 (943,262 45x45), variable: GVL.fb_loading.roller_x.roller.err, style: Lamp-Lamp1-Red
    Label (864,238 200x26), "error"
    Line (810,120) (1359,120)
    Button (1046,215 120x60), "JOG FW", colour toggle: GVL.fb_loading.roller_x.roller.forward
        OnMouseDown: execute { GVL.fb_loading.roller_x.roller.forward	:= TRUE; }
        OnMouseUp: execute { GVL.fb_loading.roller_x.roller.forward	:= FALSE; }
    Button (1045,296 120x60), "JOG BW", colour toggle: GVL.fb_loading.roller_x.roller.backward
        OnMouseDown: execute { GVL.fb_loading.roller_x.roller.backward	:= TRUE; }
        OnMouseUp: execute { GVL.fb_loading.roller_x.roller.backward	:= FALSE; }
    Line (808,373) (1357,373)
    Lamp1 (890,157 45x45), variable: GVL.fb_loading.roller_x.photo_sensor_mute_left.Q, style: Lamp-Lamp1-Green
    Label (811,133 200x26), "sensor_mute_left"
    Lamp1 (1274,157 45x45), variable: GVL.fb_loading.roller_x.photo_sensor_mute_right.Q, style: Lamp-Lamp1-Green
    Label (1195,133 200x26), "sensor_mute_right"
    Label (869,328 132x26), "roller_x"
    Lamp1 (1082,813 45x45), variable: GVL.fb_loading.roller_y.roller.sensor.Q, style: Lamp-Lamp1-Green
    Label (1005,789 200x26), "tote_detection"
    Lamp1 (937,651 45x45), variable: GVL.fb_loading.roller_y.roller.err, style: Lamp-Lamp1-Red
    Label (860,627 200x26), "error"
    Line (800,512) (1349,512)
    Button (1036,607 120x60), "JOG FW", colour toggle: GVL.fb_loading.roller_y.roller.forward
        OnMouseDown: execute { GVL.fb_loading.roller_y.roller.forward	:= TRUE; }
        OnMouseUp: execute { GVL.fb_loading.roller_y.roller.forward	:= FALSE; }
    Button (1035,688 120x60), "JOG BW", colour toggle: GVL.fb_loading.roller_y.roller.backward
        OnMouseDown: execute { GVL.fb_loading.roller_y.roller.backward	:= TRUE; }
        OnMouseUp: execute { GVL.fb_loading.roller_y.roller.backward	:= FALSE; }
    Line (800,861) (1349,861)
    Lamp1 (916,549 45x45), variable: GVL.fb_loading.roller_y.photo_sensor[0].Q, style: Lamp-Lamp1-Green
    Label (839,525 200x26), "photosensor[0]"
    Lamp1 (1240,549 45x45), variable: GVL.fb_loading.roller_y.photo_sensor[1].Q, style: Lamp-Lamp1-Green
    Label (1163,525 200x26), "photosensor[1]"
    Label (874,777 132x26), "roller_y"
    Button (1666,137 153x60), "Flood Light", colour toggle: GVL.fb_loading.floodlight
        toggle GVL.fb_loading.floodlight
        OnMouseDown: execute {  }
        OnMouseUp: execute {  }
END_VISUALIZATION

// ---- VISUs/VISUs/v_io_working.TcVIS
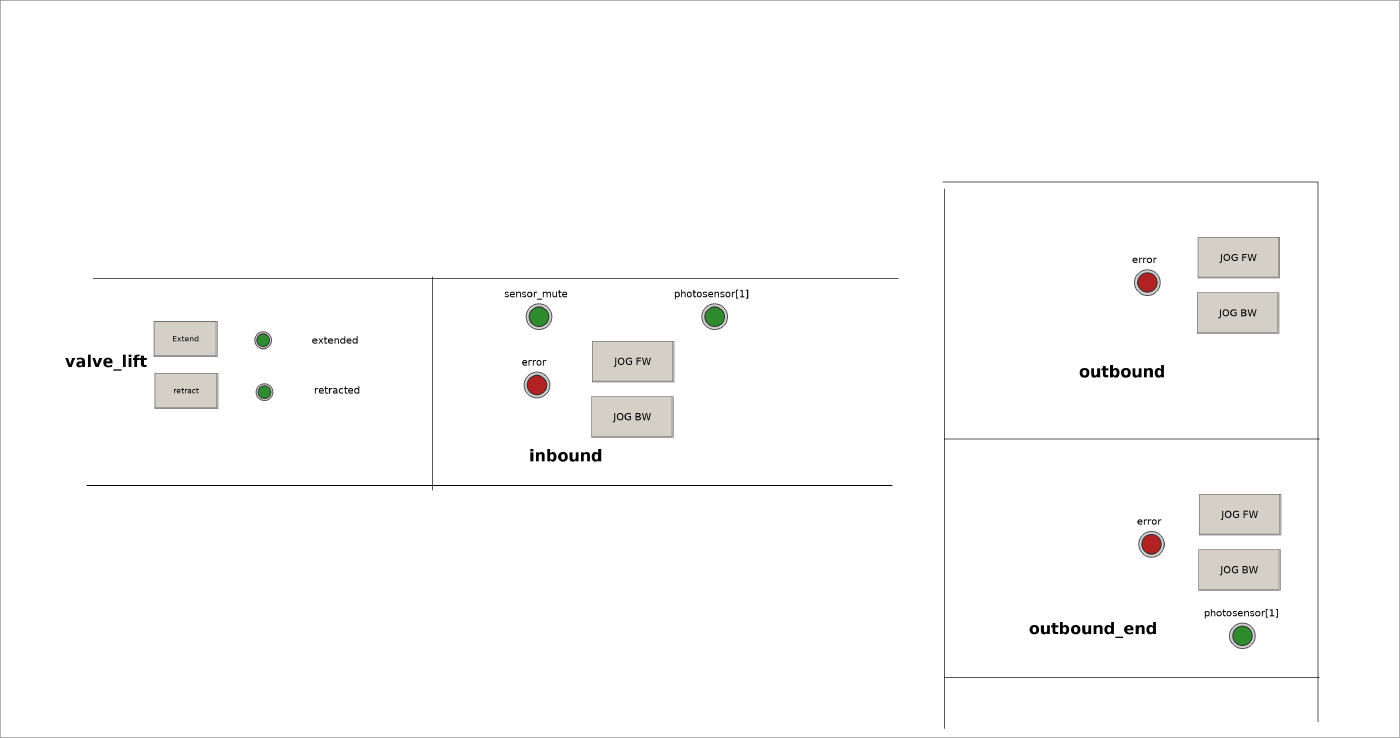
VISUALIZATION v_io_working  // 2048x1080
    Label (55,516 200x26), "valve_lift"
    Button (225,470 93x52), "Extend", colour toggle: GVL.fb_working.valve_lift.extend
        OnMouseDown: execute { GVL.fb_working.valve_lift.extend := TRUE; GVL.fb_working.valve_lift.retract := FALSE; }
    Button (226,546 93x52), "retract", colour toggle: GVL.fb_working.valve_lift.retract
        OnMouseDown: execute { GVL.fb_working.valve_lift.extend 	:= FALSE; GVL.fb_working.valve_lift.retract 	:= TRUE; }
    Lamp1 (370,483 30x30), variable: GVL.fb_working.valve_lift.extended, style: Lamp-Lamp1-Green
    Lamp1 (372,559 30x30), variable: GVL.fb_working.valve_lift.retracted, style: Lamp-Lamp1-Green
    Label (424,485 132x26), "extended"
    Label (427,558 132x26), "retracted"
    Lamp1 (763,541 45x45), variable: GVL.fb_working.roller_inbound.roller.err, style: Lamp-Lamp1-Red
    Label (681,517 200x26), "error"
    Line (136,407) (1314,407)
    Button (866,499 120x60), "JOG FW", colour toggle: GVL.fb_working.roller_inbound.roller.forward
        OnMouseDown: execute { GVL.fb_working.roller_inbound.roller.forward	:= TRUE; }
        OnMouseUp: execute { GVL.fb_working.roller_inbound.roller.forward	:= FALSE; }
    Button (865,580 120x60), "JOG BW", colour toggle: GVL.fb_working.roller_inbound.roller.backward
        OnMouseDown: execute { GVL.fb_working.roller_inbound.roller.backward	:= TRUE; }
        OnMouseUp: execute { GVL.fb_working.roller_inbound.roller.backward	:= FALSE; }
    Lamp1 (766,441 45x45), variable: GVL.fb_working.roller_inbound.photo_sensor_mute.Q, style: Lamp-Lamp1-Green
    Label (684,417 200x26), "sensor_mute"
    Lamp1 (1023,441 45x45), variable: GVL.fb_working.roller_inbound.photo_sensor.Q, style: Lamp-Lamp1-Green
    Label (941,417 200x26), "photosensor[1]"
    Label (728,654 200x26), "inbound"
    Lamp1 (1656,391 45x45), variable: GVL.fb_working.roller_outbound.roller.err, style: Lamp-Lamp1-Red
    Label (1574,367 200x26), "error"
    Line (1379,266) (1928,266)
    Button (1752,347 120x60), "JOG FW", colour toggle: GVL.fb_working.roller_outbound.roller.forward
        OnMouseDown: execute { GVL.fb_working.roller_outbound.roller.forward	:= TRUE; }
        OnMouseUp: execute { GVL.fb_working.roller_outbound.roller.forward	:= FALSE; }
    Button (1751,428 120x60), "JOG BW", colour toggle: GVL.fb_working.roller_outbound.roller.backward
        OnMouseDown: execute { GVL.fb_working.roller_outbound.roller.backward	:= TRUE; }
        OnMouseUp: execute { GVL.fb_working.roller_outbound.roller.backward	:= FALSE; }
    Lamp1 (1795,908 45x45), variable: GVL.fb_working.roller_outbound.photo_sensor.Q, style: Lamp-Lamp1-Green
    Label (1716,884 200x26), "photosensor[1]"
    Label (1542,531 200x26), "outbound"
    Lamp1 (1662,774 45x45), variable: GVL.fb_working.roller_outbound_end.roller.err, style: Lamp-Lamp1-Red
    Label (1581,750 200x26), "error"
    Line (1381,642) (1930,642)
    Button (1754,723 120x60), "JOG FW", colour toggle: GVL.fb_working.roller_outbound_end.roller.forward
        OnMouseDown: execute { GVL.fb_working.roller_outbound_end.roller.forward	:= TRUE; }
        OnMouseUp: execute { GVL.fb_working.roller_outbound_end.roller.forward	:= FALSE; }
    Button (1753,804 120x60), "JOG BW", colour toggle: GVL.fb_working.roller_outbound_end.roller.backward
        OnMouseDown: execute { GVL.fb_working.roller_outbound_end.roller.backward	:= TRUE; }
        OnMouseUp: execute { GVL.fb_working.roller_outbound_end.roller.backward	:= FALSE; }
    Line (1381,991) (1930,991)
    Label (1499,907 200x26), "outbound_end"
    Line (633,717) (633,405)
    Line (1928,1056) (1928,266)
    Line (1382,1066) (1382,276)
    Line (127,710) (1305,710)
END_VISUALIZATION
